ACTION S100_Waiting_for_Start_action:
(* @TEXT_IMPLEMENTATION := 'ST' *)
;
END_ACTION

ACTION S200_AutomaticMode_action:
_FBD_ (* Function Block Diagram *)
_END_FBD_
END_ACTION

ACTION S300_XYZ_PICKnPLACE_SFC_entry:
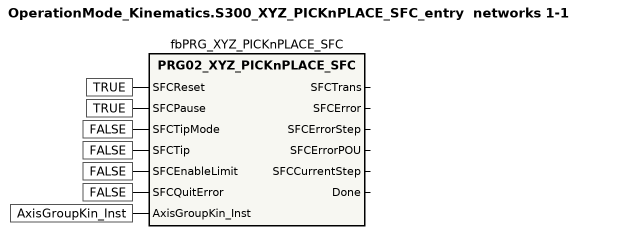
[picture p10: OperationMode_Kinematics.S300_XYZ_PICKnPLACE_SFC_entry (FBD) networks 1-1]
_FBD_ (* Function Block Diagram *)
NETWORK 1
	fbPRG_XYZ_PICKnPLACE_SFC:PRG02_XYZ_PICKnPLACE_SFC(SFCReset: TRUE, SFCPause: TRUE, SFCTipMode: FALSE, SFCTip: FALSE, SFCEnableLimit: FALSE, SFCQuitError: FALSE, AxisGroupKin_Inst: AxisGroupKin_Inst)
_END_FBD_
(* the same logic as Structured Text *)
(* Network 1 *)
fbPRG_XYZ_PICKnPLACE_SFC(SFCReset := TRUE, SFCPause := TRUE, SFCTipMode := FALSE, SFCTip := FALSE, SFCEnableLimit := FALSE, SFCQuitError := FALSE, AxisGroupKin_Inst := AxisGroupKin_Inst);
END_ACTION

ACTION S300_XYZ_PICKnPLACE_SFC_action:
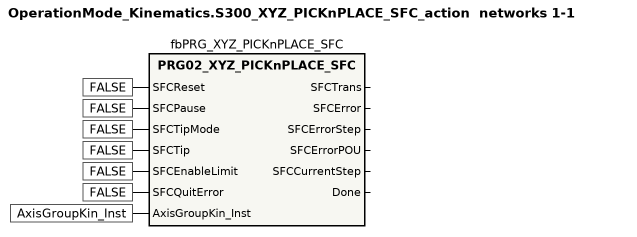
_FBD_ (* Function Block Diagram *)
NETWORK 1
	fbPRG_XYZ_PICKnPLACE_SFC:PRG02_XYZ_PICKnPLACE_SFC(SFCReset: FALSE, SFCPause: FALSE, SFCTipMode: FALSE, SFCTip: FALSE, SFCEnableLimit: FALSE, SFCQuitError: FALSE, AxisGroupKin_Inst: AxisGroupKin_Inst)
_END_FBD_
(* the same logic as Structured Text *)
(* Network 1 *)
fbPRG_XYZ_PICKnPLACE_SFC(SFCReset := FALSE, SFCPause := FALSE, SFCTipMode := FALSE, SFCTip := FALSE, SFCEnableLimit := FALSE, SFCQuitError := FALSE, AxisGroupKin_Inst := AxisGroupKin_Inst);
END_ACTION

ACTION S350_XYZ_TARG_LIN_CIRC_ST_entry:
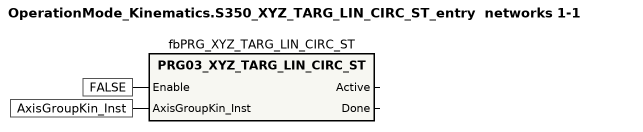
_FBD_ (* Function Block Diagram *)
NETWORK 1
	fbPRG_XYZ_TARG_LIN_CIRC_ST:PRG03_XYZ_TARG_LIN_CIRC_ST(Enable: FALSE, AxisGroupKin_Inst: AxisGroupKin_Inst)
_END_FBD_
(* the same logic as Structured Text *)
(* Network 1 *)
fbPRG_XYZ_TARG_LIN_CIRC_ST(Enable := FALSE, AxisGroupKin_Inst := AxisGroupKin_Inst);
END_ACTION

ACTION S350_XYZ_TARG_LIN_CIRC_ST_action:
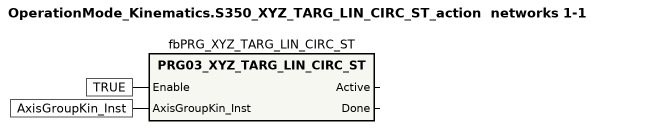
_FBD_ (* Function Block Diagram *)
NETWORK 1
	fbPRG_XYZ_TARG_LIN_CIRC_ST:PRG03_XYZ_TARG_LIN_CIRC_ST(Enable: TRUE, AxisGroupKin_Inst: AxisGroupKin_Inst)
_END_FBD_
(* the same logic as Structured Text *)
(* Network 1 *)
fbPRG_XYZ_TARG_LIN_CIRC_ST(Enable := TRUE, AxisGroupKin_Inst := AxisGroupKin_Inst);
END_ACTION

ACTION S400_XYZ_TARG_LIN_CIRC_SFC_entry:
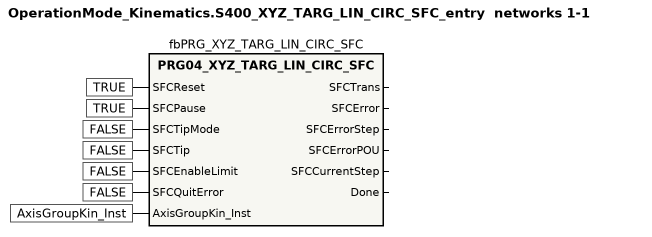
_FBD_ (* Function Block Diagram *)
NETWORK 1
	fbPRG_XYZ_TARG_LIN_CIRC_SFC:PRG04_XYZ_TARG_LIN_CIRC_SFC(SFCReset: TRUE, SFCPause: TRUE, SFCTipMode: FALSE, SFCTip: FALSE, SFCEnableLimit: FALSE, SFCQuitError: FALSE, AxisGroupKin_Inst: AxisGroupKin_Inst)
_END_FBD_
(* the same logic as Structured Text *)
(* Network 1 *)
fbPRG_XYZ_TARG_LIN_CIRC_SFC(SFCReset := TRUE, SFCPause := TRUE, SFCTipMode := FALSE, SFCTip := FALSE, SFCEnableLimit := FALSE, SFCQuitError := FALSE, AxisGroupKin_Inst := AxisGroupKin_Inst);
END_ACTION

ACTION S400_XYZ_TARG_LIN_CIRC_SFC_action:
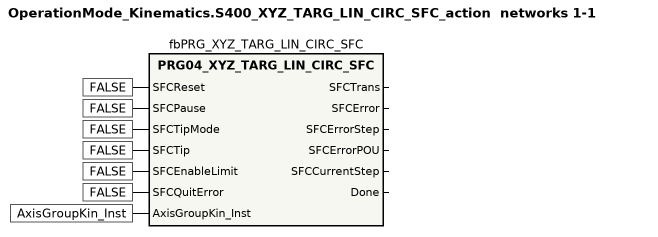
_FBD_ (* Function Block Diagram *)
NETWORK 1
	fbPRG_XYZ_TARG_LIN_CIRC_SFC:PRG04_XYZ_TARG_LIN_CIRC_SFC(SFCReset: FALSE, SFCPause: FALSE, SFCTipMode: FALSE, SFCTip: FALSE, SFCEnableLimit: FALSE, SFCQuitError: FALSE, AxisGroupKin_Inst: AxisGroupKin_Inst)
_END_FBD_
(* the same logic as Structured Text *)
(* Network 1 *)
fbPRG_XYZ_TARG_LIN_CIRC_SFC(SFCReset := FALSE, SFCPause := FALSE, SFCTipMode := FALSE, SFCTip := FALSE, SFCEnableLimit := FALSE, SFCQuitError := FALSE, AxisGroupKin_Inst := AxisGroupKin_Inst);
END_ACTION

ACTION S450_XYZ_USER_ST_entry:
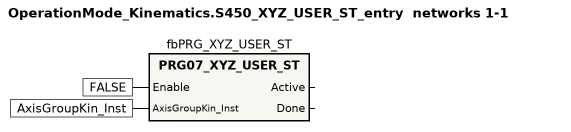
_FBD_ (* Function Block Diagram *)
NETWORK 1
	fbPRG_XYZ_USER_ST:PRG07_XYZ_USER_ST(Enable: FALSE, AxisGroupKin_Inst: AxisGroupKin_Inst)
_END_FBD_
(* the same logic as Structured Text *)
(* Network 1 *)
fbPRG_XYZ_USER_ST(Enable := FALSE, AxisGroupKin_Inst := AxisGroupKin_Inst);
END_ACTION

ACTION S450_XYZ_USER_ST_action:
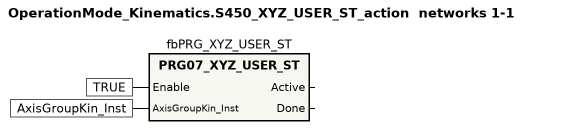
_FBD_ (* Function Block Diagram *)
NETWORK 1
	fbPRG_XYZ_USER_ST:PRG07_XYZ_USER_ST(Enable: TRUE, AxisGroupKin_Inst: AxisGroupKin_Inst)
_END_FBD_
(* the same logic as Structured Text *)
(* Network 1 *)
fbPRG_XYZ_USER_ST(Enable := TRUE, AxisGroupKin_Inst := AxisGroupKin_Inst);
END_ACTION

ACTION S500_XYZ_USER_SFC_entry:
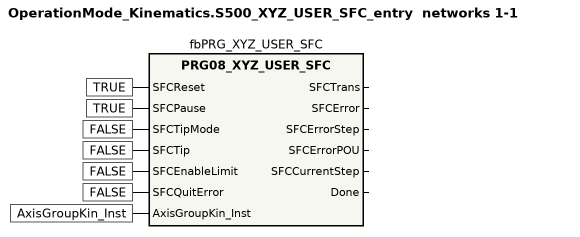
_FBD_ (* Function Block Diagram *)
NETWORK 1
	fbPRG_XYZ_USER_SFC:PRG08_XYZ_USER_SFC(SFCReset: TRUE, SFCPause: TRUE, SFCTipMode: FALSE, SFCTip: FALSE, SFCEnableLimit: FALSE, SFCQuitError: FALSE, AxisGroupKin_Inst: AxisGroupKin_Inst)
_END_FBD_
(* the same logic as Structured Text *)
(* Network 1 *)
fbPRG_XYZ_USER_SFC(SFCReset := TRUE, SFCPause := TRUE, SFCTipMode := FALSE, SFCTip := FALSE, SFCEnableLimit := FALSE, SFCQuitError := FALSE, AxisGroupKin_Inst := AxisGroupKin_Inst);
END_ACTION

ACTION S500_XYZ_USER_SFC_action:
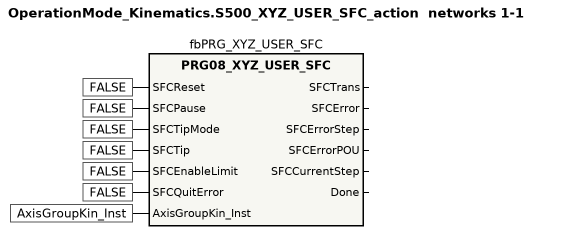
_FBD_ (* Function Block Diagram *)
NETWORK 1
	fbPRG_XYZ_USER_SFC:PRG08_XYZ_USER_SFC(SFCReset: FALSE, SFCPause: FALSE, SFCTipMode: FALSE, SFCTip: FALSE, SFCEnableLimit: FALSE, SFCQuitError: FALSE, AxisGroupKin_Inst: AxisGroupKin_Inst)
_END_FBD_
(* the same logic as Structured Text *)
(* Network 1 *)
fbPRG_XYZ_USER_SFC(SFCReset := FALSE, SFCPause := FALSE, SFCTipMode := FALSE, SFCTip := FALSE, SFCEnableLimit := FALSE, SFCQuitError := FALSE, AxisGroupKin_Inst := AxisGroupKin_Inst);
END_ACTION

ACTION S550_XYZ_FillQueue_LIN3D_with_Array_ST_entry:
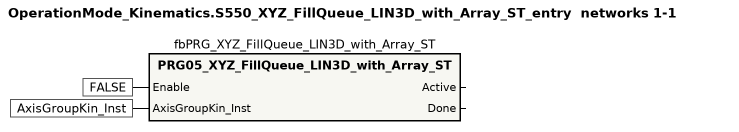
_FBD_ (* Function Block Diagram *)
NETWORK 1
	fbPRG_XYZ_FillQueue_LIN3D_with_Array_ST:PRG05_XYZ_FillQueue_LIN3D_with_Array_ST(Enable: FALSE, AxisGroupKin_Inst: AxisGroupKin_Inst)
_END_FBD_
(* the same logic as Structured Text *)
(* Network 1 *)
fbPRG_XYZ_FillQueue_LIN3D_with_Array_ST(Enable := FALSE, AxisGroupKin_Inst := AxisGroupKin_Inst);
END_ACTION

ACTION S550_XYZ_FillQueue_LIN3D_with_Array_ST_action:
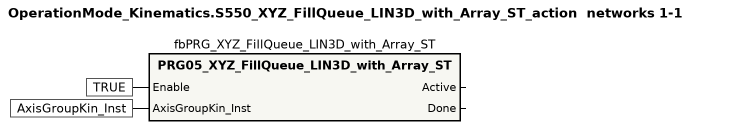
_FBD_ (* Function Block Diagram *)
NETWORK 1
	fbPRG_XYZ_FillQueue_LIN3D_with_Array_ST:PRG05_XYZ_FillQueue_LIN3D_with_Array_ST(Enable: TRUE, AxisGroupKin_Inst: AxisGroupKin_Inst)
_END_FBD_
(* the same logic as Structured Text *)
(* Network 1 *)
fbPRG_XYZ_FillQueue_LIN3D_with_Array_ST(Enable := TRUE, AxisGroupKin_Inst := AxisGroupKin_Inst);
END_ACTION

ACTION S600_XYZ_FillQueue_LIN3D_with_Array_SFC_entry:
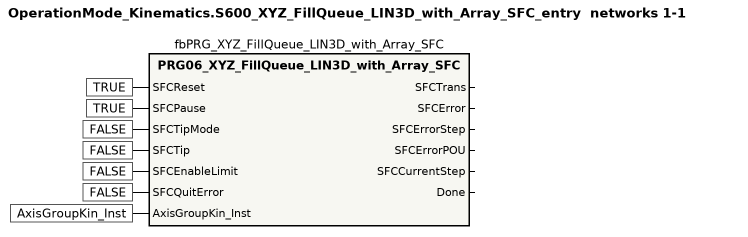
_FBD_ (* Function Block Diagram *)
NETWORK 1
	fbPRG_XYZ_FillQueue_LIN3D_with_Array_SFC:PRG06_XYZ_FillQueue_LIN3D_with_Array_SFC(SFCReset: TRUE, SFCPause: TRUE, SFCTipMode: FALSE, SFCTip: FALSE, SFCEnableLimit: FALSE, SFCQuitError: FALSE, AxisGroupKin_Inst: AxisGroupKin_Inst)
_END_FBD_
(* the same logic as Structured Text *)
(* Network 1 *)
fbPRG_XYZ_FillQueue_LIN3D_with_Array_SFC(SFCReset := TRUE, SFCPause := TRUE, SFCTipMode := FALSE, SFCTip := FALSE, SFCEnableLimit := FALSE, SFCQuitError := FALSE, AxisGroupKin_Inst := AxisGroupKin_Inst);
END_ACTION

ACTION S600_XYZ_FillQueue_LIN3D_with_Array_SFC_action:
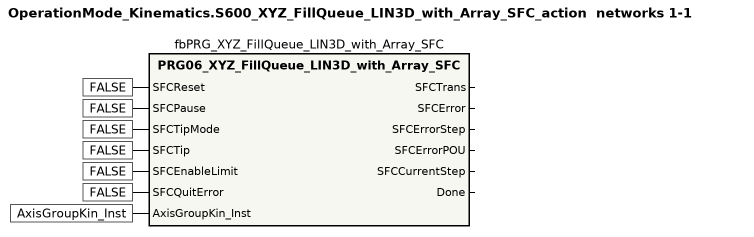
_FBD_ (* Function Block Diagram *)
NETWORK 1
	fbPRG_XYZ_FillQueue_LIN3D_with_Array_SFC:PRG06_XYZ_FillQueue_LIN3D_with_Array_SFC(SFCReset: FALSE, SFCPause: FALSE, SFCTipMode: FALSE, SFCTip: FALSE, SFCEnableLimit: FALSE, SFCQuitError: FALSE, AxisGroupKin_Inst: AxisGroupKin_Inst)
_END_FBD_
(* the same logic as Structured Text *)
(* Network 1 *)
fbPRG_XYZ_FillQueue_LIN3D_with_Array_SFC(SFCReset := FALSE, SFCPause := FALSE, SFCTipMode := FALSE, SFCTip := FALSE, SFCEnableLimit := FALSE, SFCQuitError := FALSE, AxisGroupKin_Inst := AxisGroupKin_Inst);
END_ACTION

ACTION S250_XYZ_PICKnPLACE_ST_entry:
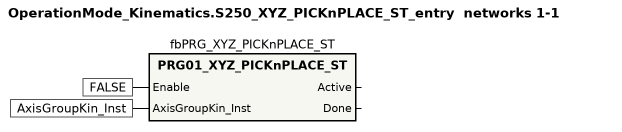
_FBD_ (* Function Block Diagram *)
NETWORK 1
	fbPRG_XYZ_PICKnPLACE_ST:PRG01_XYZ_PICKnPLACE_ST(Enable: FALSE, AxisGroupKin_Inst: AxisGroupKin_Inst)
_END_FBD_
(* the same logic as Structured Text *)
(* Network 1 *)
fbPRG_XYZ_PICKnPLACE_ST(Enable := FALSE, AxisGroupKin_Inst := AxisGroupKin_Inst);
END_ACTION

ACTION S250_XYZ_PICKnPLACE_ST_action:
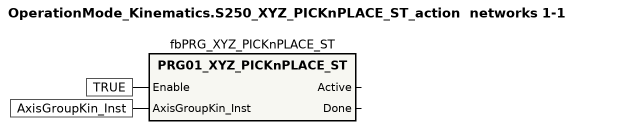
_FBD_ (* Function Block Diagram *)
NETWORK 1
	fbPRG_XYZ_PICKnPLACE_ST:PRG01_XYZ_PICKnPLACE_ST(Enable: TRUE, AxisGroupKin_Inst: AxisGroupKin_Inst)
_END_FBD_
(* the same logic as Structured Text *)
(* Network 1 *)
fbPRG_XYZ_PICKnPLACE_ST(Enable := TRUE, AxisGroupKin_Inst := AxisGroupKin_Inst);
END_ACTION

TRANSITION NOT referenced:
_FBD_ (* Function Block Diagram *)
NETWORK 1
	AND(AxisGroupKin_Inst.Out.General.Inverter.Connected[0], NOT AxisGroupKin_Inst.Out.General.Inverter.Referenced[0])
_END_FBD_
END_TRANSITION

TRANSITION referenced:
_FBD_ (* Function Block Diagram *)
NETWORK 1
	AND(AxisGroupKin_Inst.Out.General.Inverter.Connected[0], AxisGroupKin_Inst.Out.General.Inverter.Referenced[0])
_END_FBD_
END_TRANSITION

TRANSITION Homing done:
_FBD_ (* Function Block Diagram *)
NETWORK 1
	AND(AxisGroupKin_Inst.Out.General.Inverter.Connected[0], AxisGroupKin_Inst.Out.General.Inverter.Referenced[0])
_END_FBD_
END_TRANSITION

TRANSITION Automatic Mode:
_FBD_ (* Function Block Diagram *)
NETWORK 1
	AxisGroupKin_Inst.Out.General.Kin.Ready
_END_FBD_
(* the same logic as Structured Text *)
(* Network 1 *)
Automatic_Mode := AxisGroupKin_Inst.Out.General.Kin.Ready;
END_TRANSITION

TRANSITION Jog Mode:
_FBD_ (* Function Block Diagram *)
NETWORK 1
	NOT FALSE
_END_FBD_
(* the same logic as Structured Text *)
(* Network 1 *)
Jog_Mode := NOT FALSE;
END_TRANSITION

TRANSITION no Jog Mode:
_FBD_ (* Function Block Diagram *)
NETWORK 1
	FALSE
_END_FBD_
(* the same logic as Structured Text *)
(* Network 1 *)
no_Jog_Mode := FALSE;
END_TRANSITION

TRANSITION Start AND Enabled:
_FBD_ (* Function Block Diagram *)
NETWORK 1
	AND(TRUE, AxisGroupKin_Inst.Out.General.Kin.Ready)
_END_FBD_
END_TRANSITION

TRANSITION PRG1_Pick_and_Place_ST:
_FBD_ (* Function Block Diagram *)
NETWORK 1
	EQ(gKinExamples_Control[InstanceNumber].ProgramNumber, 1)
_END_FBD_
END_TRANSITION

TRANSITION Pick_and_Place_SFC:
_FBD_ (* Function Block Diagram *)
NETWORK 1
	EQ(gKinExamples_Control[InstanceNumber].ProgramNumber, 2)
_END_FBD_
END_TRANSITION

TRANSITION new Mode or Done:
_FBD_ (* Function Block Diagram *)
NETWORK 1
	OR(NE(gKinExamples_Control[InstanceNumber].ProgramNumber, 2), fbPRG_XYZ_PICKnPLACE_SFC.Done)
_END_FBD_
END_TRANSITION

TRANSITION XYZ_TARG_LIN_CIRC_ST:
_FBD_ (* Function Block Diagram *)
NETWORK 1
	EQ(gKinExamples_Control[InstanceNumber].ProgramNumber, 3)
_END_FBD_
END_TRANSITION

TRANSITION new Mode or Done:
_FBD_ (* Function Block Diagram *)
NETWORK 1
	OR(NE(gKinExamples_Control[InstanceNumber].ProgramNumber, 3), fbPRG_XYZ_TARG_LIN_CIRC_ST.Done)
_END_FBD_
END_TRANSITION

TRANSITION XYZ_TARG_LIN_CIRC_SFC:
_FBD_ (* Function Block Diagram *)
NETWORK 1
	EQ(gKinExamples_Control[InstanceNumber].ProgramNumber, 4)
_END_FBD_
END_TRANSITION

TRANSITION new Mode or Done:
_FBD_ (* Function Block Diagram *)
NETWORK 1
	OR(NE(gKinExamples_Control[InstanceNumber].ProgramNumber, 4), fbPRG_XYZ_TARG_LIN_CIRC_SFC.Done)
_END_FBD_
END_TRANSITION

TRANSITION XYZ_USER_ST:
_FBD_ (* Function Block Diagram *)
NETWORK 1
	EQ(gKinExamples_Control[InstanceNumber].ProgramNumber, 7)
_END_FBD_
END_TRANSITION

TRANSITION new Mode or Done:
_FBD_ (* Function Block Diagram *)
NETWORK 1
	OR(NE(gKinExamples_Control[InstanceNumber].ProgramNumber, 7), fbPRG_XYZ_USER_ST.Done)
_END_FBD_
END_TRANSITION

TRANSITION XYZ_USER_SFC:
_FBD_ (* Function Block Diagram *)
NETWORK 1
	EQ(gKinExamples_Control[InstanceNumber].ProgramNumber, 8)
_END_FBD_
END_TRANSITION

TRANSITION new Mode or Done:
_FBD_ (* Function Block Diagram *)
NETWORK 1
	OR(NE(gKinExamples_Control[InstanceNumber].ProgramNumber, 8), fbPRG_XYZ_USER_SFC.Done)
_END_FBD_
END_TRANSITION

TRANSITION FillQueue_LIN3D_with_Array_ST:
_FBD_ (* Function Block Diagram *)
NETWORK 1
	EQ(gKinExamples_Control[InstanceNumber].ProgramNumber, 5)
_END_FBD_
END_TRANSITION

TRANSITION new Mode or Done:
_FBD_ (* Function Block Diagram *)
NETWORK 1
	OR(NE(gKinExamples_Control[InstanceNumber].ProgramNumber, 5), fbPRG_XYZ_FillQueue_LIN3D_with_Array_ST.Done)
_END_FBD_
END_TRANSITION

TRANSITION FillQueue_LIN3D_with_Array_SFC:
_FBD_ (* Function Block Diagram *)
NETWORK 1
	EQ(gKinExamples_Control[InstanceNumber].ProgramNumber, 6)
_END_FBD_
END_TRANSITION

TRANSITION new Mode OR Done:
_FBD_ (* Function Block Diagram *)
NETWORK 1
	OR(NE(gKinExamples_Control[InstanceNumber].ProgramNumber, 6), fbPRG_XYZ_FillQueue_LIN3D_with_Array_SFC.Done)
_END_FBD_
END_TRANSITION

TRANSITION Jog Mode:
_FBD_ (* Function Block Diagram *)
NETWORK 1
	NOT FALSE
_END_FBD_
(* the same logic as Structured Text *)
(* Network 1 *)
Jog_Mode := NOT FALSE;
END_TRANSITION

TRANSITION new Mode or Done:
_FBD_ (* Function Block Diagram *)
NETWORK 1
	OR(NE(gKinExamples_Control[InstanceNumber].ProgramNumber, 1), fbPRG_XYZ_PICKnPLACE_ST.Done)
_END_FBD_
END_TRANSITION
END_FUNCTION_BLOCK

(* POU AxisGroupControl_Kinematics/Examples/PRG01_XYZ_PICKnPLACE_ST, ST *)
(*##############################################################################################################

	IMPORTANT NOTICE:
 	This example is a special and free service that demonstrates only the basic 
	approach to generating a PLC program as a non-binding sample. 
	SEW is not liable for the contents of the sample program.

	Name:			PRG_XYZ_PICKnPLACE_ST
	Job:			Example program		
					Sequence: XYZ_PICKnPLACE_P2 -> P3 -> P4 -> P3 -> P2 -> P1
					
################################################################################################################*)
FUNCTION_BLOCK  PRG01_XYZ_PICKnPLACE_ST
VAR_INPUT
	Enable : BOOL;
END_VAR
VAR_OUTPUT
	Active : BOOL;
	Done : BOOL;
END_VAR
VAR
	nState : INT := 0;
	fbRtrig : R_TRIG;
	i : INT;
END_VAR
VAR_IN_OUT
	AxisGroupKin_Inst											: ST_AxisGroupKin_Instance;
END_VAR
(* Initialisation at rising edge of VAR_INPUT Enable *)
fbRtrig(CLK:=Enable);
IF fbRtrig.Q THEN
	nState := 0;
	Active := TRUE;
END_IF

(* No execution, if Enable = False *)
IF (Enable = FALSE) THEN
	Done := FALSE;
	RETURN;
END_IF


CASE nState OF
0:	(*Start*)
	IF AxisGroupKin.ConfigDataAvailable THEN
		nState := 5;
	END_IF

5:	(* Up *)
	(* Initialize Kinematic Flags*)
	AxisGroupKin_Inst.In.Cp.Settings.PlusTargetCartABC:=FALSE;
	AxisGroupKin_Inst.In.Cp.Settings.UseMasterPosition:=FALSE;

(* TARGET_CART settings *)
	(* Motion Parameters *)
	AxisGroupKin_Inst.In.Target.Cart.Velocity := CART_VEL100;
	AxisGroupKin_Inst.In.Target.Cart.Acceleration := CART_ACC100;
	AxisGroupKin_Inst.In.Target.Cart.Deceleration := CART_DEC100;
	AxisGroupKin_Inst.In.Target.Cart.Jerk:=CART_Jerk100;
	AxisGroupKin_Inst.In.Target.Synchronization:= KIN_NO_SYNC;
	(* Coordinate System *)
	AxisGroupKin_Inst.In.Target.CoordSys:=KIN_KCS;

	AxisGroupKin_Inst.In.General.Mode := KIN_TARGET_CART;

	AxisGroupKin_Inst.In.Target.Position := XYZ_PICKnPLACE_P2;

	IF (MC_KinInProximity(Threshold := XYZ_PICKnPLACE_BlendingDistance,
			Position := AxisGroupKin_Inst.In.Target.Position,
			CoordSys := AxisGroupKin_Inst.In.Target.CoordSys,
			Dimension := 2#0000_0111, ActPos := AxisGroupKin_Inst.Out.General.Position)) THEN
		nState := 10;
	END_IF
	AxisGroupKin_Inst.In.Simu3D.Ctrl.Pen_TCP_WCS:=TRUE;

10:	(* Side *)
	AxisGroupKin_Inst.In.Target.Position := XYZ_PICKnPLACE_P3;
	IF (MC_KinInProximity(Threshold := XYZ_PICKnPLACE_BlendingDistance,
			Position := AxisGroupKin_Inst.In.Target.Position,
			CoordSys := AxisGroupKin_Inst.In.Target.CoordSys,
			Dimension := 2#0000_0111, ActPos := AxisGroupKin_Inst.Out.General.Position)) THEN
		nState := 20;
	END_IF

20:	(* Down *)
	AxisGroupKin_Inst.In.Target.Position := XYZ_PICKnPLACE_P4;
	IF (MC_KinInProximity(Threshold := 0.0,
			Position := AxisGroupKin_Inst.In.Target.Position,
			CoordSys := AxisGroupKin_Inst.In.Target.CoordSys,
			Dimension := 2#0000_0111, ActPos := AxisGroupKin_Inst.Out.General.Position)
			AND AxisGroupKin_Inst.Out.General.Standstill.ActCoordSys) THEN
		nState :=30;
	END_IF

30:	(* Up *)
	AxisGroupKin_Inst.In.Target.Position := XYZ_PICKnPLACE_P3;
	IF (MC_KinInProximity(Threshold := XYZ_PICKnPLACE_BlendingDistance,
			Position := AxisGroupKin_Inst.In.Target.Position,
			CoordSys := AxisGroupKin_Inst.In.Target.CoordSys,
			Dimension := 2#0000_0111, ActPos := AxisGroupKin_Inst.Out.General.Position)) THEN
		nState := 40;
	END_IF

40:	(* Side *)
	AxisGroupKin_Inst.In.Target.Position := XYZ_PICKnPLACE_P2;
	IF (MC_KinInProximity(Threshold := XYZ_PICKnPLACE_BlendingDistance,
			Position := AxisGroupKin_Inst.In.Target.Position,
			CoordSys := AxisGroupKin_Inst.In.Target.CoordSys,
			Dimension := 2#0000_0111, ActPos := AxisGroupKin_Inst.Out.General.Position)) THEN
		nState := 50;
	END_IF

50:	(* Down *)
	AxisGroupKin_Inst.In.Target.Position := XYZ_PICKnPLACE_P1;
	IF (MC_KinInProximity(Threshold := 0.0,
			Position := AxisGroupKin_Inst.In.Target.Position,
			CoordSys := AxisGroupKin_Inst.In.Target.CoordSys,
			Dimension := 2#0000_0111, ActPos := AxisGroupKin_Inst.Out.General.Position)
			AND AxisGroupKin_Inst.Out.General.Standstill.ActCoordSys) THEN
		AxisGroupKin_Inst.In.Simu3D.Ctrl.Pen_TCP_WCS:=FALSE;
		Done := TRUE;
		Active := FALSE;
	END_IF

ELSE
;

END_CASE
END_FUNCTION_BLOCK

(* POU AxisGroupControl_Kinematics/Examples/PRG02_XYZ_PICKnPLACE_SFC, SFC *)
(*##############################################################################################################

	IMPORTANT NOTICE:
 	This example is a special and free service that demonstrates only the basic 
	approach to generating a PLC program as a non-binding sample. 
	SEW is not liable for the contents of the sample program.

	Name:			PRG_XYZ_PICKnPLACE_SFC
	Job:			Example program		
					Sequence: XYZ_PICKnPLACE_P2 -> P3 -> P4 -> P3 -> P2 -> P1	

################################################################################################################*)
FUNCTION_BLOCK PRG02_XYZ_PICKnPLACE_SFC
VAR_INPUT
	SFCReset:BOOL;
	(*SFCInit:BOOL;*)
	SFCPause:BOOL;

	SFCTipMode:BOOL;
	SFCTip:BOOL;
	SFCEnableLimit:BOOL;
	SFCQuitError:BOOL;
END_VAR
VAR_OUTPUT
	SFCTrans:BOOL;
	SFCError:BOOL;
	SFCErrorStep:STRING;
	SFCErrorPOU:STRING;
	SFCCurrentStep:STRING;
	Done:BOOL;
END_VAR
VAR

END_VAR
VAR_IN_OUT
	AxisGroupKin_Inst											: ST_AxisGroupKin_Instance;
END_VAR
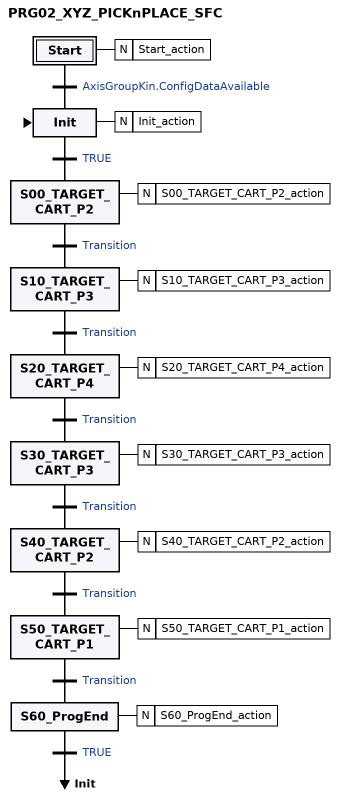
INITIAL_STEP Start:
	Start_action(N);
END_STEP
TRANSITION FROM Start TO Init := AxisGroupKin.ConfigDataAvailable;
END_TRANSITION
STEP Init:
	Init_action(N);
END_STEP
TRANSITION FROM Init TO S00_TARGET_CART_P2 := TRUE;
END_TRANSITION
STEP S00_TARGET_CART_P2:
	S00_TARGET_CART_P2_action(N);
END_STEP
TRANSITION FROM S00_TARGET_CART_P2 TO S10_TARGET_CART_P3 := Transition;
END_TRANSITION
STEP S10_TARGET_CART_P3:
	S10_TARGET_CART_P3_action(N);
END_STEP
TRANSITION FROM S10_TARGET_CART_P3 TO S20_TARGET_CART_P4 := Transition;
END_TRANSITION
STEP S20_TARGET_CART_P4:
	S20_TARGET_CART_P4_action(N);
END_STEP
TRANSITION FROM S20_TARGET_CART_P4 TO S30_TARGET_CART_P3 := Transition;
END_TRANSITION
STEP S30_TARGET_CART_P3:
	S30_TARGET_CART_P3_action(N);
END_STEP
TRANSITION FROM S30_TARGET_CART_P3 TO S40_TARGET_CART_P2 := Transition;
END_TRANSITION
STEP S40_TARGET_CART_P2:
	S40_TARGET_CART_P2_action(N);
END_STEP
TRANSITION FROM S40_TARGET_CART_P2 TO S50_TARGET_CART_P1 := Transition;
END_TRANSITION
STEP S50_TARGET_CART_P1:
	S50_TARGET_CART_P1_action(N);
END_STEP
TRANSITION FROM S50_TARGET_CART_P1 TO S60_ProgEnd := Transition;
END_TRANSITION
STEP S60_ProgEnd:
	S60_ProgEnd_action(N);
END_STEP
TRANSITION FROM S60_ProgEnd TO Init := TRUE;
END_TRANSITION

ACTION Start_action:
Done:=FALSE;
END_ACTION

ACTION Init_action:
(* Initialize Kinematic Flags*)
	AxisGroupKin_Inst.In.Cp.Settings.PlusTargetCartABC:=FALSE;
	AxisGroupKin_Inst.In.Cp.Settings.UseMasterPosition:=FALSE;

(* TARGET_CART settings *)
	(* Motion Parameters *)
	AxisGroupKin_Inst.In.Target.Cart.Velocity := CART_VEL100;
	AxisGroupKin_Inst.In.Target.Cart.Acceleration := CART_ACC100;
	AxisGroupKin_Inst.In.Target.Cart.Deceleration := CART_DEC100;
	AxisGroupKin_Inst.In.Target.Cart.Jerk := CART_Jerk100;
	AxisGroupKin_Inst.In.Target.Synchronization := KIN_NO_SYNC;
	(* Coordinate System *)
	AxisGroupKin_Inst.In.Target.CoordSys := KIN_KCS;

	AxisGroupKin_Inst.In.General.Mode := KIN_TARGET_CART;
END_ACTION

ACTION S00_TARGET_CART_P2_action:
AxisGroupKin_Inst.In.Target.Position := XYZ_PICKnPLACE_P2;
END_ACTION

ACTION S10_TARGET_CART_P3_action:
AxisGroupKin_Inst.In.Target.Position := XYZ_PICKnPLACE_P3;
END_ACTION

ACTION S20_TARGET_CART_P4_action:
AxisGroupKin_Inst.In.Target.Position := XYZ_PICKnPLACE_P4;
END_ACTION

ACTION S30_TARGET_CART_P3_action:
AxisGroupKin_Inst.In.Target.Position := XYZ_PICKnPLACE_P3;
END_ACTION

ACTION S40_TARGET_CART_P2_action:
AxisGroupKin_Inst.In.Target.Position := XYZ_PICKnPLACE_P2;
END_ACTION

ACTION S50_TARGET_CART_P1_action:
AxisGroupKin_Inst.In.Target.Position := XYZ_PICKnPLACE_P1;
END_ACTION

ACTION S60_ProgEnd_action:
Done:=TRUE;
END_ACTION

TRANSITION Transition:
MC_KinInProximity(Threshold := XYZ_PICKnPLACE_BlendingDistance,
			Position := AxisGroupKin_Inst.In.Target.Position,
			CoordSys := AxisGroupKin_Inst.In.Target.CoordSys,
			Dimension := 2#0000_0111, ActPos := AxisGroupKin_Inst.Out.General.Position)
END_TRANSITION

TRANSITION Transition:
MC_KinInProximity(Threshold := XYZ_PICKnPLACE_BlendingDistance,
			Position := AxisGroupKin_Inst.In.Target.Position,
			CoordSys := AxisGroupKin_Inst.In.Target.CoordSys,
			Dimension := 2#0000_0111, ActPos := AxisGroupKin_Inst.Out.General.Position)
END_TRANSITION

TRANSITION Transition:
MC_KinInProximity(Threshold := 0.0,
			Position := AxisGroupKin_Inst.In.Target.Position,
			CoordSys := AxisGroupKin_Inst.In.Target.CoordSys,
			Dimension := 2#0000_0111, ActPos := AxisGroupKin_Inst.Out.General.Position)
AND
AxisGroupKin_Inst.Out.General.Standstill.ActCoordSys
END_TRANSITION

TRANSITION Transition:
MC_KinInProximity(Threshold := XYZ_PICKnPLACE_BlendingDistance,
			Position := AxisGroupKin_Inst.In.Target.Position,
			CoordSys := AxisGroupKin_Inst.In.Target.CoordSys,
			Dimension := 2#0000_0111, ActPos := AxisGroupKin_Inst.Out.General.Position)
END_TRANSITION

TRANSITION Transition:
MC_KinInProximity(Threshold := XYZ_PICKnPLACE_BlendingDistance,
			Position := AxisGroupKin_Inst.In.Target.Position,
			CoordSys := AxisGroupKin_Inst.In.Target.CoordSys,
			Dimension := 2#0000_0111, ActPos := AxisGroupKin_Inst.Out.General.Position)
END_TRANSITION

TRANSITION Transition:
MC_KinInProximity(Threshold := 0.0,
			Position := AxisGroupKin_Inst.In.Target.Position,
			CoordSys := AxisGroupKin_Inst.In.Target.CoordSys,
			Dimension := 2#0000_0111, ActPos := AxisGroupKin_Inst.Out.General.Position)
AND
AxisGroupKin_Inst.Out.General.Standstill.ActCoordSys
END_TRANSITION
END_FUNCTION_BLOCK

(* POU AxisGroupControl_Kinematics/Examples/PRG03_XYZ_TARG_LIN_CIRC_ST, ST *)
(*##############################################################################################################

	IMPORTANT NOTICE:
 	This example is a special and free service that demonstrates only the basic 
	approach to generating a PLC program as a non-binding sample. 
	SEW is not liable for the contents of the sample program.

	Name:			PRG_XYZ_TARG_LIN_CIRC_ST
	Job:			Example program			
					Sequence: TARGET_CART to XYZ_TARG_LIN_CIRC_P1 -> LIN_XY to P2 -> CIRC_XZ with R3/A3 -> LIN_3D to P4 -> LIN_XY to P1

################################################################################################################*)
FUNCTION_BLOCK PRG03_XYZ_TARG_LIN_CIRC_ST
VAR_INPUT
	Enable : BOOL;
END_VAR
VAR_OUTPUT
	Active : BOOL;
	Done : BOOL;
END_VAR
VAR
	nState : INT;
	fbRtrig : R_TRIG;
END_VAR
VAR_IN_OUT
	AxisGroupKin_Inst											: ST_AxisGroupKin_Instance;
END_VAR
(* Initialisation at rising edge of VAR_INPUT Enable *)
fbRtrig(CLK:=Enable);
IF fbRtrig.Q THEN
	nState	:= 0;
	Active := TRUE;
END_IF

(* No execution, if Enable = False *)
IF NOT Enable THEN
	Done := FALSE;
	RETURN;
END_IF


CASE nState OF
0:	(*Start*)
	IF AxisGroupKin.ConfigDataAvailable THEN
		nState := 5;
	END_IF
5:	(* TARGET_CART to XYZ_TARG_LIN_CIRC_P1 *)
	(* Initialize Kinematic Flags*)
	AxisGroupKin_Inst.In.Cp.Settings.PlusTargetCartABC:=FALSE;
	AxisGroupKin_Inst.In.Cp.Settings.UseMasterPosition:=FALSE;

(* TARGET_CART settings *)
	(* Motion Parameters *)
	AxisGroupKin_Inst.In.Target.Cart.Acceleration := CART_ACC50;
	AxisGroupKin_Inst.In.Target.Cart.Deceleration := CART_DEC50;
	AxisGroupKin_Inst.In.Target.Cart.Velocity := CART_VEL50;
	AxisGroupKin_Inst.In.Target.Cart.Jerk:=CART_Jerk100;
	AxisGroupKin_Inst.In.Target.Synchronization:= KIN_NO_SYNC;
	(* Coordinate System *)
	AxisGroupKin_Inst.In.Target.CoordSys:=KIN_KCS;

	AxisGroupKin_Inst.In.General.Mode := KIN_TARGET_CART;

	AxisGroupKin_Inst.In.Target.Position := XYZ_TARG_LIN_CIRC_P1;
	IF (MC_KinInProximity(Threshold := 0.0,
			Position := AxisGroupKin_Inst.In.Target.Position,
			CoordSys := AxisGroupKin_Inst.In.Target.CoordSys,
			Dimension := 2#0000_0111, ActPos := AxisGroupKin_Inst.Out.General.Position)
			AND AxisGroupKin_Inst.Out.General.Standstill.ActCoordSys) THEN
		nState := 10;
	END_IF

10:	(* Straight line to XYZ_TARG_LIN_CIRC_P2, as soon as XYZ_TARG_LIN_CIRC_P1 has been reached *)

		AxisGroupKin_Inst.In.General.Mode := KIN_LIN_XY;
		AxisGroupKin_Inst.In.Cp.Segment.Position := XYZ_TARG_LIN_CIRC_P2;
(* CP motion parameters *)
		(* settings for whole path / all segments *)
		AxisGroupKin_Inst.In.Cp.Path.VelocityPercentage:=100;
		AxisGroupKin_Inst.In.Cp.Path.FidelityPercentage :=100;
		(* Settings for the segment, which should be added to the queue *)
		AxisGroupKin_Inst.In.Cp.Segment.Translation.Velocity := 1000;
		AxisGroupKin_Inst.In.Cp.Segment.Translation.Acceleration := 100;
		AxisGroupKin_Inst.In.Cp.Segment.Translation.Deceleration := 100;
		AxisGroupKin_Inst.In.Cp.Segment.Translation.Jerk := 100;
		AxisGroupKin_Inst.In.Cp.Segment.Blending.Distance := 50;
		AxisGroupKin_Inst.In.Cp.Segment.Blending.LimitationPercentage := 50;

		AxisGroupKin_Inst.In.Cp.Segment.ID := AxisGroupKin_Inst.In.Cp.Segment.ID + 1;	(* Change the SegmentID to add the segment to the queue *)

		AxisGroupKin_Inst.In.Simu3D.Ctrl.Pen_TCP_WCS := TRUE;

		nState := 20;

20:	(* A circle section is written into the queue directly after the straight line *)
	IF (AxisGroupKin_Inst.Out.Cp.Queue.LastMappedSegID = AxisGroupKin_Inst.In.Cp.Segment.ID) THEN (* Wait until the segment was added to the queue; this is not required if FB_KinControl is executed in the same task *)
		AxisGroupKin_Inst.In.General.Mode := KIN_CIRC_ZX;
		(* Parameters to define the circle *)
		AxisGroupKin_Inst.In.Cp.Segment.Circ.Mode := KIN_RADIUS_ANGLE;	(* Define the circle with the radius and angle *)
		AxisGroupKin_Inst.In.Cp.Segment.Circ.Direction := KIN_CW;	(* Draw circle ClockWise *)
		AxisGroupKin_Inst.In.Cp.Segment.Circ.Radius := XYZ_TARG_LIN_CIRC_R3;
		AxisGroupKin_Inst.In.Cp.Segment.Circ.Angle := XYZ_TARG_LIN_CIRC_A3;


		AxisGroupKin_Inst.In.Cp.Segment.ID := AxisGroupKin_Inst.In.Cp.Segment.ID + 1;
		nState := 30;
	END_IF

30:	(* A Straight line to XYZ_TARG_LIN_CIRC_P4 is written into the queue directly after the circle section
		-> Blending to the straight line is performed automatically *)
	IF (AxisGroupKin_Inst.Out.Cp.Queue.LastMappedSegID = AxisGroupKin_Inst.In.Cp.Segment.ID) THEN
		AxisGroupKin_Inst.In.General.Mode := KIN_LIN_3D;
		AxisGroupKin_Inst.In.Cp.Segment.Position := XYZ_TARG_LIN_CIRC_P4;


		AxisGroupKin_Inst.In.Cp.Segment.ID := AxisGroupKin_Inst.In.Cp.Segment.ID + 1;
		nState := 40;
	END_IF

40:	(* Straight line to XYZ_TARG_LIN_CIRC_P1 is written into the queue directly after the previous straight line
		-> Blending to the straight line is performed automatically *)
	IF (AxisGroupKin_Inst.Out.Cp.Queue.LastMappedSegID = AxisGroupKin_Inst.In.Cp.Segment.ID) THEN
		AxisGroupKin_Inst.In.General.Mode := KIN_LIN_XY;
		AxisGroupKin_Inst.In.Cp.Segment.Position := XYZ_TARG_LIN_CIRC_P1;


		AxisGroupKin_Inst.In.Cp.Segment.ID := AxisGroupKin_Inst.In.Cp.Segment.ID + 1;
		nState := 50;
	END_IF

50:	(* Program end, as soon as XYZ_TARG_LIN_CIRC_P1 has been reached *)
	IF (AxisGroupKin_Inst.Out.Cp.Path.EndReached)
	AND (AxisGroupKin_Inst.Out.Cp.Queue.LastMappedSegID = AxisGroupKin_Inst.In.Cp.Segment.ID) THEN
		Done := TRUE;
		Active := FALSE;
		AxisGroupKin_Inst.In.Simu3D.Ctrl.Pen_TCP_WCS := FALSE;
	END_IF

ELSE
;

END_CASE
END_FUNCTION_BLOCK

(* POU AxisGroupControl_Kinematics/Examples/PRG04_XYZ_TARG_LIN_CIRC_SFC, SFC *)
(*##############################################################################################################

	IMPORTANT NOTICE:
 	This example is a special and free service that demonstrates only the basic 
	approach to generating a PLC program as a non-binding sample. 
	SEW is not liable for the contents of the sample program.

	Name:			PRG_XYZ_TARG_LIN_CIRC_SFC
	Job:			Example program			
					Sequence: TARGET_CART to XYZ_TARG_LIN_CIRC_P1 -> LIN_XY to P2 -> CIRC_XZ with R3/A3 -> LIN_3D to P4 -> LIN_XY to P1

################################################################################################################*)
FUNCTION_BLOCK PRG04_XYZ_TARG_LIN_CIRC_SFC
VAR_INPUT
	SFCReset:BOOL;
	(*SFCInit:BOOL;*)
	SFCPause:BOOL;

	SFCTipMode:BOOL;
	SFCTip:BOOL;
	SFCEnableLimit:BOOL;
	SFCQuitError:BOOL;

END_VAR
VAR_OUTPUT
	SFCTrans:BOOL;
	SFCError:BOOL;
	SFCErrorStep:STRING;
	SFCErrorPOU:STRING;
(*	SFCErrorAnalyzation:STRING;*)
	SFCCurrentStep:STRING;
	Done:BOOL;
END_VAR
VAR

END_VAR
VAR_IN_OUT
	AxisGroupKin_Inst											: ST_AxisGroupKin_Instance;
END_VAR
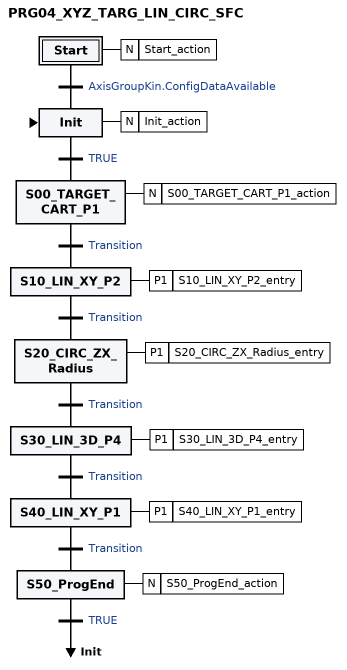
INITIAL_STEP Start:
	Start_action(N);
END_STEP
TRANSITION FROM Start TO Init := AxisGroupKin.ConfigDataAvailable;
END_TRANSITION
STEP Init:
	Init_action(N);
END_STEP
TRANSITION FROM Init TO S00_TARGET_CART_P1 := TRUE;
END_TRANSITION
STEP S00_TARGET_CART_P1:
	S00_TARGET_CART_P1_action(N);
END_STEP
TRANSITION FROM S00_TARGET_CART_P1 TO S10_LIN_XY_P2 := Transition;
END_TRANSITION
STEP S10_LIN_XY_P2:
	S10_LIN_XY_P2_entry(P1);
END_STEP
TRANSITION FROM S10_LIN_XY_P2 TO S20_CIRC_ZX_Radius := Transition;
END_TRANSITION
STEP S20_CIRC_ZX_Radius:
	S20_CIRC_ZX_Radius_entry(P1);
END_STEP
TRANSITION FROM S20_CIRC_ZX_Radius TO S30_LIN_3D_P4 := Transition;
END_TRANSITION
STEP S30_LIN_3D_P4:
	S30_LIN_3D_P4_entry(P1);
END_STEP
TRANSITION FROM S30_LIN_3D_P4 TO S40_LIN_XY_P1 := Transition;
END_TRANSITION
STEP S40_LIN_XY_P1:
	S40_LIN_XY_P1_entry(P1);
END_STEP
TRANSITION FROM S40_LIN_XY_P1 TO S50_ProgEnd := Transition;
END_TRANSITION
STEP S50_ProgEnd:
	S50_ProgEnd_action(N);
END_STEP
TRANSITION FROM S50_ProgEnd TO Init := TRUE;
END_TRANSITION

ACTION Start_action:
Done:=FALSE;
END_ACTION

ACTION Init_action:
(* Initialize Kinematic Flags*)
	AxisGroupKin_Inst.In.Cp.Settings.PlusTargetCartABC:=FALSE;
	AxisGroupKin_Inst.In.Cp.Settings.UseMasterPosition:=FALSE;

(* TARGET_CART settings *)
	(* Motion Parameters *)
	AxisGroupKin_Inst.In.Target.Cart.Acceleration := CART_ACC50;
	AxisGroupKin_Inst.In.Target.Cart.Deceleration := CART_DEC50;
	AxisGroupKin_Inst.In.Target.Cart.Velocity := CART_VEL50;
	AxisGroupKin_Inst.In.Target.Cart.Jerk:=CART_Jerk100;
	AxisGroupKin_Inst.In.Target.Synchronization:= KIN_NO_SYNC;
	(* Coordinate System *)
	AxisGroupKin_Inst.In.Target.CoordSys:=KIN_KCS;

	AxisGroupKin_Inst.In.General.Mode := KIN_TARGET_CART;
END_ACTION

ACTION S00_TARGET_CART_P1_action:
AxisGroupKin_Inst.In.Target.Position :=  XYZ_TARG_LIN_CIRC_P1;
END_ACTION

ACTION S10_LIN_XY_P2_entry:
(* Straight line to XYZ_TARG_LIN_CIRC_P2, as soon as XYZ_TARG_LIN_CIRC_P1 has been reached *)

		AxisGroupKin_Inst.In.General.Mode := KIN_LIN_XY;
		AxisGroupKin_Inst.In.Cp.Segment.Position := XYZ_TARG_LIN_CIRC_P2;
(* CP motion parameters *)
		(* settings for whole path / all segments *)
		AxisGroupKin_Inst.In.Cp.Path.VelocityPercentage:=100;
		AxisGroupKin_Inst.In.Cp.Path.FidelityPercentage :=100;
		(* Settings for the segment, which should be added to the queue *)
		AxisGroupKin_Inst.In.Cp.Segment.Translation.Velocity := 1000;
		AxisGroupKin_Inst.In.Cp.Segment.Translation.Acceleration := 100;
		AxisGroupKin_Inst.In.Cp.Segment.Translation.Deceleration := 100;
		AxisGroupKin_Inst.In.Cp.Segment.Translation.Jerk := 100;
		AxisGroupKin_Inst.In.Cp.Segment.Blending.Distance := 50;
		AxisGroupKin_Inst.In.Cp.Segment.Blending.LimitationPercentage := 50;

		AxisGroupKin_Inst.In.Cp.Segment.ID := AxisGroupKin_Inst.In.Cp.Segment.ID + 1;	(* Change the SegmentID to add the segment to the queue *)

		AxisGroupKin_Inst.In.Simu3D.Ctrl.Pen_TCP_WCS := TRUE;
END_ACTION

ACTION S20_CIRC_ZX_Radius_entry:
AxisGroupKin_Inst.In.General.Mode := KIN_CIRC_ZX;
(* Parameters to define the circle *)
AxisGroupKin_Inst.In.Cp.Segment.Circ.Mode := KIN_RADIUS_ANGLE;	(* Define the circle with the radius and angle *)
AxisGroupKin_Inst.In.Cp.Segment.Circ.Direction := KIN_CW;	(* Draw circle ClockWise *)
AxisGroupKin_Inst.In.Cp.Segment.Circ.Radius := XYZ_TARG_LIN_CIRC_R3;
AxisGroupKin_Inst.In.Cp.Segment.Circ.Angle := XYZ_TARG_LIN_CIRC_A3;


AxisGroupKin_Inst.In.Cp.Segment.ID := AxisGroupKin_Inst.In.Cp.Segment.ID + 1;
END_ACTION

ACTION S30_LIN_3D_P4_entry:
AxisGroupKin_Inst.In.General.Mode := KIN_LIN_3D;
AxisGroupKin_Inst.In.Cp.Segment.Position := XYZ_TARG_LIN_CIRC_P4;


AxisGroupKin_Inst.In.Cp.Segment.ID := AxisGroupKin_Inst.In.Cp.Segment.ID + 1;
END_ACTION

ACTION S40_LIN_XY_P1_entry:
AxisGroupKin_Inst.In.General.Mode := KIN_LIN_XY;
AxisGroupKin_Inst.In.Cp.Segment.Position := XYZ_TARG_LIN_CIRC_P1;


AxisGroupKin_Inst.In.Cp.Segment.ID := AxisGroupKin_Inst.In.Cp.Segment.ID + 1;
END_ACTION

ACTION S50_ProgEnd_action:
Done := TRUE;
AxisGroupKin_Inst.In.Simu3D.Ctrl.Pen_TCP_WCS := FALSE;  (* Process Off *)
END_ACTION

TRANSITION Transition:
MC_KinInProximity(Threshold := 0.0,
			Position := AxisGroupKin_Inst.In.Target.Position,
			CoordSys := AxisGroupKin_Inst.In.Target.CoordSys,
			Dimension := 2#0000_0111, ActPos := AxisGroupKin_Inst.Out.General.Position)
AND
AxisGroupKin_Inst.Out.General.Standstill.ActCoordSys
END_TRANSITION

TRANSITION Transition:
(* Wait until the segment was added to the queue; this is not required if FB_KinControl is executed in the same task *)
AxisGroupKin_Inst.Out.Cp.Queue.LastMappedSegID = AxisGroupKin_Inst.In.Cp.Segment.ID
END_TRANSITION

TRANSITION Transition:
(* Wait until the segment was added to the queue; this is not required if FB_KinControl is executed in the same task *)
AxisGroupKin_Inst.Out.Cp.Queue.LastMappedSegID = AxisGroupKin_Inst.In.Cp.Segment.ID
END_TRANSITION

TRANSITION Transition:
(* Wait until the segment was added to the queue; this is not required if FB_KinControl is executed in the same task *)
AxisGroupKin_Inst.Out.Cp.Queue.LastMappedSegID = AxisGroupKin_Inst.In.Cp.Segment.ID
END_TRANSITION

TRANSITION Transition:
(AxisGroupKin_Inst.Out.Cp.Path.EndReached) AND
(AxisGroupKin_Inst.Out.Cp.Queue.LastMappedSegID = AxisGroupKin_Inst.In.Cp.Segment.ID)
END_TRANSITION
END_FUNCTION_BLOCK

(* POU AxisGroupControl_Kinematics/Examples/PRG05_XYZ_FillQueue_LIN3D_with_Array_ST, ST *)
(*##############################################################################################################

	IMPORTANT NOTICE:
 	This example is a special and free service that demonstrates only the basic 
	approach to generating a PLC program as a non-binding sample. 
	SEW is not liable for the contents of the sample program.

	Name:			PRG_XYZ_FillQueue_LIN3D_with_Array_ST
	Job:			Example program			

################################################################################################################*)
FUNCTION_BLOCK PRG05_XYZ_FillQueue_LIN3D_with_Array_ST

VAR_INPUT
	Enable: BOOL;
END_VAR
VAR_OUTPUT
	Active: BOOL;
	Done: BOOL;
END_VAR
VAR
	nState : INT := 0;
	i:INT:=1;
END_VAR
VAR_IN_OUT
	AxisGroupKin_Inst											: ST_AxisGroupKin_Instance;
END_VAR
IF NOT Enable THEN
	Done:=FALSE;
	Active := FALSE;
	i:=1;
	nState:=0;
	RETURN;
END_IF
CASE nState OF
0:	(*Start*)
	IF AxisGroupKin.ConfigDataAvailable THEN
		nState := 5;
	END_IF

5:	(* Initialization and TARGET_CART to last point in queue *)

	(* Initialize kinematics flags*)
	AxisGroupKin_Inst.In.Cp.Settings.PlusTargetCartABC :=FALSE;
	AxisGroupKin_Inst.In.Cp.Settings.UseMasterPosition:=FALSE;

(* CP settings *)
	(* Initialize SegID *)
	AxisGroupKin_Inst.In.Cp.Segment.ID := AxisGroupKin_Inst.Out.Cp.Queue.LastMappedSegID;
	(* Initialize global point array *)
	points[1].x:=10;	points[1].y:=100;	points[1].z:=50;
	points[2].x:=10;	points[2].y:=200;	points[2].z:=100;
	points[3].x:=50;	points[3].y:=300;	points[3].z:=50;
	points[4].x:=100;	points[4].y:=350;	points[4].z:=100;
	points[5].x:=200;	points[5].y:=300;	points[5].z:=50;
	points[6].x:=300;	points[6].y:=200;	points[6].z:=100;
	points[7].x:=300;	points[7].y:=100;	points[7].z:=50;
	points[8].x:=200;	points[8].y:=50;	points[8].z:=100;
	points[9].x:=100;	points[9].y:=10;	points[9].z:=50;
	points[10].x:=50;	points[10].y:=50;	points[10].z:=100;
	(* motion parameters for CP modes *)
	AxisGroupKin_Inst.In.Cp.Segment.Translation.Velocity := 100;
	AxisGroupKin_Inst.In.Cp.Segment.Translation.Acceleration := 100;
	AxisGroupKin_Inst.In.Cp.Segment.Translation.Deceleration := 100;
	AxisGroupKin_Inst.In.Cp.Segment.Translation.Jerk := 100;
	AxisGroupKin_Inst.In.Cp.Segment.Blending.Distance := 30;
	AxisGroupKin_Inst.In.Cp.Segment.Blending.LimitationPercentage := 50;
	AxisGroupKin_Inst.In.Cp.Segment.Mode := KIN_CONTINUOUS_PATH;
	AxisGroupKin_Inst.In.Cp.Path.VelocityPercentage:=100;
	AxisGroupKin_Inst.In.Cp.Path.FidelityPercentage :=100;

(* TARGET_CART settings *)
	(* Set motion parameters for target mode*)
	AxisGroupKin_Inst.In.Target.Cart.Acceleration := CART_ACC50;
	AxisGroupKin_Inst.In.Target.Cart.Deceleration := CART_DEC50;
	AxisGroupKin_Inst.In.Target.Cart.Velocity := CART_VEL50;
	AxisGroupKin_Inst.In.Target.Cart.Jerk:=CART_Jerk100;
	AxisGroupKin_Inst.In.Target.CoordSys := KIN_KCS;
	AxisGroupKin_Inst.In.Target.Synchronization:= KIN_NO_SYNC;
	(* move to last point in array *)
	AxisGroupKin_Inst.In.Target.Position[1] := points[10].x;
	AxisGroupKin_Inst.In.Target.Position[2] := points[10].y;
	AxisGroupKin_Inst.In.Target.Position[3] := points[10].z;

	AxisGroupKin_Inst.In.General.Mode := KIN_TARGET_CART;

	IF (MC_KinInProximity(Threshold := 0.0,
			Position := AxisGroupKin_Inst.In.Target.Position,
			CoordSys := AxisGroupKin_Inst.In.Target.CoordSys,
			Dimension := 2#0000_0111, ActPos := AxisGroupKin_Inst.Out.General.Position)
			AND AxisGroupKin_Inst.Out.General.Standstill.ActCoordSys) THEN
		nState := 10;
	END_IF
10:	(*Fill Queue *)
	IF i <=10 THEN
		AxisGroupKin_Inst.In.Simu3D.Ctrl.Pen_TCP_WCS :=TRUE;
		IF AxisGroupKin_Inst.Out.Cp.Queue.LastMappedSegID = AxisGroupKin_Inst.In.Cp.Segment.ID THEN
			AxisGroupKin_Inst.In.General.Mode := KIN_LIN_3D;
			AxisGroupKin_Inst.In.Cp.Segment.Position[1] := points[i].x;
			AxisGroupKin_Inst.In.Cp.Segment.Position[2] := points[i].y;
			AxisGroupKin_Inst.In.Cp.Segment.Position[3] := points[i].z;
			AxisGroupKin_Inst.In.Cp.Segment.ID := AxisGroupKin_Inst.In.Cp.Segment.ID + 1;
			i:=i+1;
		END_IF
	ELSIF AxisGroupKin_Inst.Out.Cp.Path.EndReached THEN
		Done := TRUE;
		Active := FALSE;
		AxisGroupKin_Inst.In.Simu3D.Ctrl.Pen_TCP_WCS := FALSE;
	END_IF
END_CASE
END_FUNCTION_BLOCK

(* POU AxisGroupControl_Kinematics/Examples/PRG06_XYZ_FillQueue_LIN3D_with_Array_SFC, SFC *)
(*##############################################################################################################

	IMPORTANT NOTICE:
 	This example is a special and free service that demonstrates only the basic 
	approach to generating a PLC program as a non-binding sample. 
	SEW is not liable for the contents of the sample program.

	Name:			PRG_XYZ_FillQueue_LIN3D_with_Array_SFC
	Job:			Example program		

################################################################################################################*)
FUNCTION_BLOCK PRG06_XYZ_FillQueue_LIN3D_with_Array_SFC
VAR_INPUT
	SFCReset:BOOL;
	(*SFCInit:BOOL;*)
	SFCPause:BOOL;

	SFCTipMode:BOOL;
	SFCTip:BOOL;
	SFCEnableLimit:BOOL;
	SFCQuitError:BOOL;

END_VAR
VAR_OUTPUT
	SFCTrans:BOOL;
	SFCError:BOOL;
	SFCErrorStep:STRING;
	SFCErrorPOU:STRING;
	SFCCurrentStep:STRING;
	Done:BOOL;
END_VAR
VAR
	i:INT;
END_VAR
VAR_IN_OUT
	AxisGroupKin_Inst	: ST_AxisGroupKin_Instance;
END_VAR
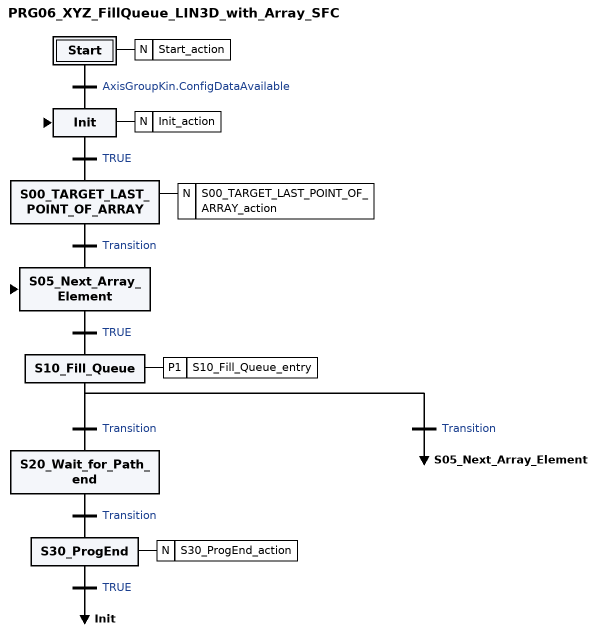
INITIAL_STEP Start:
	Start_action(N);
END_STEP
TRANSITION FROM Start TO Init := AxisGroupKin.ConfigDataAvailable;
END_TRANSITION
STEP Init:
	Init_action(N);
END_STEP
TRANSITION FROM Init TO S00_TARGET_LAST_POINT_OF_ARRAY := TRUE;
END_TRANSITION
STEP S00_TARGET_LAST_POINT_OF_ARRAY:
	S00_TARGET_LAST_POINT_OF_ARRAY_action(N);
END_STEP
TRANSITION FROM S00_TARGET_LAST_POINT_OF_ARRAY TO S05_Next_Array_Element := Transition;
END_TRANSITION
STEP S05_Next_Array_Element:
END_STEP
TRANSITION FROM S05_Next_Array_Element TO S10_Fill_Queue := TRUE;
END_TRANSITION
STEP S10_Fill_Queue:
	S10_Fill_Queue_entry(P1);
END_STEP
TRANSITION FROM S10_Fill_Queue TO S20_Wait_for_Path_end := Transition;
END_TRANSITION
TRANSITION FROM S10_Fill_Queue TO S05_Next_Array_Element := Transition;
END_TRANSITION
STEP S20_Wait_for_Path_end:
END_STEP
TRANSITION FROM S20_Wait_for_Path_end TO S30_ProgEnd := Transition;
END_TRANSITION
STEP S30_ProgEnd:
	S30_ProgEnd_action(N);
END_STEP
TRANSITION FROM S30_ProgEnd TO Init := TRUE;
END_TRANSITION

ACTION Start_action:
Done:=FALSE;
END_ACTION

ACTION Init_action:
(* Initialize kinematics flags*)
	AxisGroupKin_Inst.In.Cp.Settings.PlusTargetCartABC :=FALSE;
	AxisGroupKin_Inst.In.Cp.Settings.UseMasterPosition:=FALSE;

(* CP settings *)
	(* Initialize SegID *)
	AxisGroupKin_Inst.In.Cp.Segment.ID := AxisGroupKin_Inst.Out.Cp.Queue.LastMappedSegID;
	(* Initialize global point array *)
	points[1].x:=10;	points[1].y:=100;	points[1].z:=50;
	points[2].x:=10;	points[2].y:=200;	points[2].z:=100;
	points[3].x:=50;	points[3].y:=300;	points[3].z:=50;
	points[4].x:=100;	points[4].y:=350;	points[4].z:=100;
	points[5].x:=200;	points[5].y:=300;	points[5].z:=50;
	points[6].x:=300;	points[6].y:=200;	points[6].z:=100;
	points[7].x:=300;	points[7].y:=100;	points[7].z:=50;
	points[8].x:=200;	points[8].y:=50;	points[8].z:=100;
	points[9].x:=100;	points[9].y:=10;	points[9].z:=50;
	points[10].x:=50;	points[10].y:=50;	points[10].z:=100;
	(* motion parameters for CP modes *)
	AxisGroupKin_Inst.In.Cp.Segment.Translation.Velocity := 100;
	AxisGroupKin_Inst.In.Cp.Segment.Translation.Acceleration := 100;
	AxisGroupKin_Inst.In.Cp.Segment.Translation.Deceleration := 100;
	AxisGroupKin_Inst.In.Cp.Segment.Translation.Jerk := 100;
	AxisGroupKin_Inst.In.Cp.Segment.Blending.Distance := 30;
	AxisGroupKin_Inst.In.Cp.Segment.Blending.LimitationPercentage := 50;
	AxisGroupKin_Inst.In.Cp.Segment.Mode := KIN_CONTINUOUS_PATH;
	AxisGroupKin_Inst.In.Cp.Path.VelocityPercentage:=100;
	AxisGroupKin_Inst.In.Cp.Path.FidelityPercentage :=100;

(* TARGET_CART settings *)
	(* Set motion parameters for target mode*)
	AxisGroupKin_Inst.In.Target.Cart.Acceleration := CART_ACC50;
	AxisGroupKin_Inst.In.Target.Cart.Deceleration := CART_DEC50;
	AxisGroupKin_Inst.In.Target.Cart.Velocity := CART_VEL50;
	AxisGroupKin_Inst.In.Target.Cart.Jerk:=CART_Jerk100;
	AxisGroupKin_Inst.In.Target.CoordSys := KIN_KCS;
	AxisGroupKin_Inst.In.Target.Synchronization:= KIN_NO_SYNC;

	AxisGroupKin_Inst.In.General.Mode := KIN_TARGET_CART;

	i:=1;
END_ACTION

ACTION S00_TARGET_LAST_POINT_OF_ARRAY_action:
(* move to last point in array *)
AxisGroupKin_Inst.In.Target.Position[1] := points[10].x;
AxisGroupKin_Inst.In.Target.Position[2] := points[10].y;
AxisGroupKin_Inst.In.Target.Position[3] := points[10].z;
END_ACTION

ACTION S10_Fill_Queue_entry:
AxisGroupKin_Inst.In.General.Mode			:= KIN_LIN_3D;
AxisGroupKin_Inst.In.Cp.Segment.Position[1]	:= points[i].x;
AxisGroupKin_Inst.In.Cp.Segment.Position[2] 	:= points[i].y;
AxisGroupKin_Inst.In.Cp.Segment.Position[3] 	:= points[i].z;
AxisGroupKin_Inst.In.Cp.Segment.ID 		:= AxisGroupKin_Inst.In.Cp.Segment.ID + 1;

i:=i+1;
END_ACTION

ACTION S30_ProgEnd_action:
Done:=TRUE;
END_ACTION

TRANSITION Transition:
MC_KinInProximity(Threshold := 0.0,
			Position := AxisGroupKin_Inst.In.Target.Position,
			CoordSys := AxisGroupKin_Inst.In.Target.CoordSys,
			Dimension := 2#0000_0111, ActPos := AxisGroupKin_Inst.Out.General.Position)

AND
AxisGroupKin_Inst.Out.General.Standstill.ActCoordSys
END_TRANSITION

TRANSITION Transition:
(AxisGroupKin_Inst.Out.Cp.Queue.LastMappedSegID= AxisGroupKin_Inst.In.Cp.Segment.ID) AND (i >10)
END_TRANSITION

TRANSITION Transition:
AxisGroupKin_Inst.Out.Cp.Queue.LastMappedSegID = AxisGroupKin_Inst.In.Cp.Segment.ID
END_TRANSITION

TRANSITION Transition:
AxisGroupKin_Inst.Out.Cp.Path.EndReached
END_TRANSITION
END_FUNCTION_BLOCK

(* POU AxisGroupControl_Kinematics/Examples/PRG07_XYZ_USER_ST, ST *)
(*##############################################################################################################

	IMPORTANT NOTICE:
 	This example is a special and free service that demonstrates only the basic 
	approach to generating a PLC program as a non-binding sample. 
	SEW is not liable for the contents of the sample program.

	Name:			PRG_XYZ_USER_ST
	Job:			Example program
					Simple program, in which you can implement your own sample sequence.			

################################################################################################################*)
FUNCTION_BLOCK PRG07_XYZ_USER_ST
VAR_INPUT
	Enable : BOOL;
END_VAR
VAR_OUTPUT
	Active : BOOL;
	Done : BOOL;
END_VAR
VAR
	nState : INT;
	fbRtrig : R_TRIG;
END_VAR
VAR_IN_OUT
	AxisGroupKin_Inst											: ST_AxisGroupKin_Instance;
END_VAR
(* Initialisation at rising edge of VAR_INPUT Enable *)
fbRtrig(CLK:=Enable);
IF fbRtrig.Q THEN
	nState	:= 0;
	Active := TRUE;
END_IF

(* No execution, if Enable = False *)
IF NOT Enable THEN
	Done := FALSE;
	RETURN;
END_IF

CASE nState OF
0:	(*Start*)
	IF AxisGroupKin.ConfigDataAvailable THEN
		nState := 5;
	END_IF
5:	(* TARGET_CART to XYZ_USER_P1 *)
	(* Initialize Kinematic Flags*)
	AxisGroupKin_Inst.In.Cp.Settings.PlusTargetCartABC:=FALSE;
	AxisGroupKin_Inst.In.Cp.Settings.UseMasterPosition:=FALSE;

(* TARGET_CART settings *)
	(* Motion Parameters *)
	AxisGroupKin_Inst.In.Target.Cart.Velocity := CART_VEL50;
	AxisGroupKin_Inst.In.Target.Cart.Acceleration := CART_ACC50;
	AxisGroupKin_Inst.In.Target.Cart.Deceleration := CART_DEC50;
	AxisGroupKin_Inst.In.Target.Cart.Jerk:=CART_Jerk100;
	AxisGroupKin_Inst.In.Target.Synchronization:= KIN_NO_SYNC;
	(* Coordinate System *)
	AxisGroupKin_Inst.In.Target.CoordSys:=KIN_KCS;

	AxisGroupKin_Inst.In.General.Mode := KIN_TARGET_CART;

	AxisGroupKin_Inst.In.Simu3D.Ctrl.Pen_TCP_WCS := TRUE;  (* Process On *)

	AxisGroupKin_Inst.In.Target.Position := XYZ_USER_P1;
	IF (MC_KinInProximity(Threshold := 0.0,
			Position := AxisGroupKin_Inst.In.Target.Position,
			CoordSys := AxisGroupKin_Inst.In.Target.CoordSys,
			Dimension := 2#0000_0111, ActPos := AxisGroupKin_Inst.Out.General.Position)
			AND AxisGroupKin_Inst.Out.General.Standstill.ActCoordSys) THEN
		nState := 10;
	END_IF

10:	(* TARGET_CART to XYZ_USER_P2 *)
	AxisGroupKin_Inst.In.Target.Position := XYZ_USER_P2;
	IF (MC_KinInProximity(Threshold := 0.0,
			Position := AxisGroupKin_Inst.In.Target.Position,
			CoordSys := AxisGroupKin_Inst.In.Target.CoordSys,
			Dimension := 2#0000_0111, ActPos := AxisGroupKin_Inst.Out.General.Position)
			AND AxisGroupKin_Inst.Out.General.Standstill.ActCoordSys) THEN
		Done := TRUE;
		Active := FALSE;
		AxisGroupKin_Inst.In.Simu3D.Ctrl.Pen_TCP_WCS := FALSE;  (* Process Off *)
	END_IF

ELSE
;

END_CASE
END_FUNCTION_BLOCK

(* POU AxisGroupControl_Kinematics/Examples/PRG08_XYZ_USER_SFC, SFC *)
(*##############################################################################################################

	IMPORTANT NOTICE:
 	This example is a special and free service that demonstrates only the basic 
	approach to generating a PLC program as a non-binding sample. 
	SEW is not liable for the contents of the sample program.

	Name:			PRG_XYZ_USER_SFC
	Job:			Example program
					Simple program, in which you can implement your own sample sequence.				

################################################################################################################*)
FUNCTION_BLOCK PRG08_XYZ_USER_SFC
VAR_INPUT
	SFCReset:BOOL;
	(*SFCInit:BOOL;*)
	SFCPause:BOOL;

	SFCTipMode:BOOL;
	SFCTip:BOOL;
	SFCEnableLimit:BOOL;
	SFCQuitError:BOOL;

END_VAR
VAR_OUTPUT
	SFCTrans:BOOL;
	SFCError:BOOL;
	SFCErrorStep:STRING;
	SFCErrorPOU:STRING;
(*	SFCErrorAnalyzation:STRING;*)
	SFCCurrentStep:STRING;
	Done:BOOL;
END_VAR
VAR

END_VAR
VAR_IN_OUT
	AxisGroupKin_Inst											: ST_AxisGroupKin_Instance;
END_VAR
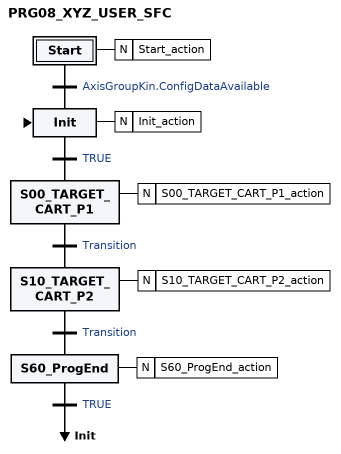
INITIAL_STEP Start:
	Start_action(N);
END_STEP
TRANSITION FROM Start TO Init := AxisGroupKin.ConfigDataAvailable;
END_TRANSITION
STEP Init:
	Init_action(N);
END_STEP
TRANSITION FROM Init TO S00_TARGET_CART_P1 := TRUE;
END_TRANSITION
STEP S00_TARGET_CART_P1:
	S00_TARGET_CART_P1_action(N);
END_STEP
TRANSITION FROM S00_TARGET_CART_P1 TO S10_TARGET_CART_P2 := Transition;
END_TRANSITION
STEP S10_TARGET_CART_P2:
	S10_TARGET_CART_P2_action(N);
END_STEP
TRANSITION FROM S10_TARGET_CART_P2 TO S60_ProgEnd := Transition;
END_TRANSITION
STEP S60_ProgEnd:
	S60_ProgEnd_action(N);
END_STEP
TRANSITION FROM S60_ProgEnd TO Init := TRUE;
END_TRANSITION

ACTION Start_action:
Done:=FALSE;
END_ACTION

ACTION Init_action:
(* Initialize Kinematic Flags*)
AxisGroupKin_Inst.In.Cp.Settings.PlusTargetCartABC:=FALSE;
AxisGroupKin_Inst.In.Cp.Settings.UseMasterPosition:=FALSE;

(* TARGET_CART settings *)
	(* Motion Parameters *)
	AxisGroupKin_Inst.In.Target.Cart.Velocity := CART_VEL50;
	AxisGroupKin_Inst.In.Target.Cart.Acceleration := CART_ACC50;
	AxisGroupKin_Inst.In.Target.Cart.Deceleration := CART_DEC50;
	AxisGroupKin_Inst.In.Target.Cart.Jerk:=CART_Jerk100;
	AxisGroupKin_Inst.In.Target.Synchronization:= KIN_NO_SYNC;
	(* Coordinate System *)
	AxisGroupKin_Inst.In.Target.CoordSys:=KIN_KCS;

AxisGroupKin_Inst.In.General.Mode := KIN_TARGET_CART;

AxisGroupKin_Inst.In.Simu3D.Ctrl.Pen_TCP_WCS := TRUE;  (* Process On *)
END_ACTION

ACTION S00_TARGET_CART_P1_action:
AxisGroupKin_Inst.In.Target.Position := XYZ_USER_P1;
END_ACTION

ACTION S10_TARGET_CART_P2_action:
AxisGroupKin_Inst.In.Target.Position := XYZ_USER_P2;
END_ACTION

ACTION S60_ProgEnd_action:
Done := TRUE;
AxisGroupKin_Inst.In.Simu3D.Ctrl.Pen_TCP_WCS := FALSE;  (* Process Off *)
END_ACTION

TRANSITION Transition:
MC_KinInProximity(Threshold := 0.0,
			Position := AxisGroupKin_Inst.In.Target.Position,
			CoordSys := AxisGroupKin_Inst.In.Target.CoordSys,
			Dimension := 2#0000_0111, ActPos := AxisGroupKin_Inst.Out.General.Position)
AND
AxisGroupKin_Inst.Out.General.Standstill.ActCoordSys
END_TRANSITION

TRANSITION Transition:
MC_KinInProximity(Threshold := 0.0,
			Position := AxisGroupKin_Inst.In.Target.Position,
			CoordSys := AxisGroupKin_Inst.In.Target.CoordSys,
			Dimension := 2#0000_0111, ActPos := AxisGroupKin_Inst.Out.General.Position)
AND
AxisGroupKin_Inst.Out.General.Standstill.ActCoordSys
END_TRANSITION
END_FUNCTION_BLOCK

(* POU PRG_Kinematics/PRG_TaskPriority_Kinematics, ST *)
PROGRAM PRG_TaskPriority_Kinematics
VAR
END_VAR
(*#######################################################################################

	PRG_TaskPriority_Kinematics

	ToDo: Call this program in the task configuration after PRG_TaskPriority();

########################################################################################*)

(* Do not remove! *)
AxisGroupControl_Priority_Kinematics();
END_PROGRAM

(* POU SewRobotLanguage/FB_SewRobotLanguage_User_Function, ST *)
(*##############################################################################################################

	IMPORTANT NOTICE:
 	This example is a special and free service that demonstrates only the basic 
	approach to generating a PLC program as a non-binding sample. 
	SEW is not liable for the contents of the sample program.

	Name:			FB_SewRobotLanguage_User_Function
	Job:			Contains User Functions that can be called in SRL Program

################################################################################################################*)
FUNCTION_BLOCK FB_SewRobotLanguage_User_Function
VAR_INPUT
	Enable								: BOOL;				(* Enable of Function*)
	NumberOfFunction				: INT;					(* Number of the Fuction what will be executed*)
	bParaValue						: BOOL;				(* Boolean	Value *)
	rParaValue						: LREAL;				(* Real 	Value *)
	posParaValue						: ST_SRL_DimPos; 	(* Position Vektor *)
	Instance							: UINT;
END_VAR
VAR_OUTPUT
	Done								: BOOL;				(* true if function is executed correctly*)
	Error								: BOOL;				(* Error Flag*)
	ErrorID								: DWORD;				(* Error ID*)
END_VAR
VAR_IN_OUT
	SRL_Dat_Var						: ST_SRL_Variables;
	AxisGroupKin_Inst				: ST_AxisGroupKin_Instance;	(*AxisGroupControl Kinematics Variable*)
END_VAR
VAR
	(*Handling Kin: Zuweisung Dynamikwerte anhand der SegParRecords*)
	nIndex 								: UINT;


	SegParaRecCart_Act				: UINT;
	SegParaRecAxis_Act				: UINT;
	SegParaRecCp_Act				: UINT;
	SegParaRecRot_Act				: UINT;
	SegParaRecTp_Act				: UINT;

	nSynchronization					: WORD;

	fbTON					: TON;
	tTime					: TIME;

	ModuleName 			: STRING(50)		:='SRL_User_Function';
	Message				: STRING(128)	:='SRL_User_Function';
	nTaskID				: WORD;
	nTaskPriority			: DINT;
END_VAR
IF ((Instance < 1) OR (Instance > KIN_AXISGROUPKIN_MAX_NUMBER_OF_KINEMATICS_INSTANCES)) THEN
	MC_MsgHandler_Enter(
		Class 		:= MSGHANDLER_CLASS_ERROR,
		Source 	:= MSGHANDLER_SOURCE_TECHNOLOGYMODULE,
		Module 	:= 'SewRobotLanguage',
		Instance 	:= Instance,
		ID 			:= E_KIN_SRL_INSTANCENUMBER_NOT_VALID,
		Text 		:= 'MC_Enter_Message_Buffer_SRL: InstanceNumber Not Valid',
		Value_n1 	:= 0 ,
		Value_n2 	:= 0,
		Value_f1 	:= 0,
		Value_f2 	:= 0,
		ErrorArchivingOnlyAfterReset := FALSE,
		ForceEntryInNewElement := FALSE);
		(*weil kein gültige Instanznummer da, hier die 1 auf Fehler setzen*)
		SRL.Inst[1].Interface.Out.FBError	:= TRUE;
		SRL.Inst[1].Interface.Out.FBErrorID	:= E_KIN_SRL_INSTANCENUMBER_NOT_VALID;

	RETURN;
END_IF

tTime:=REAL_TO_TIME(rParaValue);

fbTON(IN:=Enable , PT:=tTime );

IF Enable THEN
	CASE NumberOfFunction OF
		11:(* SegParRecAxis *)

			SegParaRecAxis_Act := LREAL_TO_UINT(rParaValue);
			IF (SegParaRecAxis_Act > 8) OR (SegParaRecAxis_Act < 1) THEN(*tbd ID festlegen*)
				Message:= ' SegParRecord Number §n1§ not valid => Init Program and Reset Error';
				MC_Enter_Message_Buffer_HandlingKin(
					E_HANDLINGKIN_SEG_PAR_RECORD_NUMBER_NOT_VALID,Message,0,0,0,0,TRUE,Instance,Error,ErrorID);
				RETURN;
			END_IF
			FOR nIndex := 1 TO 8 DO
				(*Es wird nur noch die Geschwindigkeit vom Override Percentage beeinflußt *)

				SRL_Dat_Var.PositionData.Value[SRL_SYS_IN_AXIS_VEL].Dim[nIndex]:=AxisGroupHandlingKin.Inst[Instance].Config.SegmentParameterRecord[SegParaRecAxis_Act].AxisVel[nIndex];
				SRL_Dat_Var.PositionData.Value[SRL_SYS_IN_AXIS_ACC].Dim[nIndex]:=AxisGroupHandlingKin.Inst[Instance].Config.SegmentParameterRecord[SegParaRecAxis_Act].AxisAcc[nIndex]		(** TargetVelocityPercentagefaktor*TargetVelocityPercentagefaktor*);
				SRL_Dat_Var.PositionData.Value[SRL_SYS_IN_AXIS_DEC].Dim[nIndex]:=AxisGroupHandlingKin.Inst[Instance].Config.SegmentParameterRecord[SegParaRecAxis_Act].AxisDec[nIndex]		(** TargetVelocityPercentagefaktor*TargetVelocityPercentagefaktor*);
				IF AxisGroupKin_Inst.Config.General.RealJerk_InsteadOfJerkTime THEN
					SRL_Dat_Var.PositionData.Value[SRL_SYS_IN_AXIS_JERK].Dim[nIndex]:=AxisGroupHandlingKin.Inst[Instance].Config.SegmentParameterRecord[SegParaRecAxis_Act].AxisJerk[nIndex](** TargetVelocityPercentagefaktor*TargetVelocityPercentagefaktor*TargetVelocityPercentagefaktor*);
				ELSE
					SRL_Dat_Var.PositionData.Value[SRL_SYS_IN_AXIS_JERK].Dim[nIndex]:=AxisGroupHandlingKin.Inst[Instance].Config.SegmentParameterRecord[SegParaRecAxis_Act].AxisJerk[nIndex] (*/ TargetVelocityPercentagefaktor*)	;
				END_IF
			END_FOR
			nSynchronization:=0;
			nSynchronization.1:= AxisGroupHandlingKin.Inst[Instance].Config.SegmentParameterRecord[SegParaRecAxis_Act].AxisSynchronization[1];
			nSynchronization.2:= AxisGroupHandlingKin.Inst[Instance].Config.SegmentParameterRecord[SegParaRecAxis_Act].AxisSynchronization[2];
			nSynchronization.3:= AxisGroupHandlingKin.Inst[Instance].Config.SegmentParameterRecord[SegParaRecAxis_Act].AxisSynchronization[3];
			nSynchronization.4:= AxisGroupHandlingKin.Inst[Instance].Config.SegmentParameterRecord[SegParaRecAxis_Act].AxisSynchronization[4];
			nSynchronization.5:= AxisGroupHandlingKin.Inst[Instance].Config.SegmentParameterRecord[SegParaRecAxis_Act].AxisSynchronization[5];
			nSynchronization.6:= AxisGroupHandlingKin.Inst[Instance].Config.SegmentParameterRecord[SegParaRecAxis_Act].AxisSynchronization[6];
			nSynchronization.7:= AxisGroupHandlingKin.Inst[Instance].Config.SegmentParameterRecord[SegParaRecAxis_Act].AxisSynchronization[7];
			nSynchronization.8:= AxisGroupHandlingKin.Inst[Instance].Config.SegmentParameterRecord[SegParaRecAxis_Act].AxisSynchronization[8];
			SRL_Dat_Var.RealData.Value[SRL_SYS_IN_TARGET_AXIS_SYNC]:=WORD_TO_LREAL(nSynchronization);
			Done:=TRUE;

		12:(* SegParRecCart	*)

			SegParaRecCart_Act:=LREAL_TO_UINT(rParaValue);
			IF (SegParaRecCart_Act > 8) OR (SegParaRecCart_Act < 1) THEN(*tbd ID festlegen*)
				Message:= ' SegParRecord Number §n1§ not valid => Init Program and Reset Error';
				MC_Enter_Message_Buffer_HandlingKin(
					E_HANDLINGKIN_SEG_PAR_RECORD_NUMBER_NOT_VALID,Message,0,0,0,0,TRUE,Instance,Error,ErrorID);
				RETURN;
			END_IF
			FOR nIndex := 1 TO 6 DO
				SRL_Dat_Var.PositionData.Value[SRL_SYS_IN_CART_VEL].Dim[nIndex]:=AxisGroupHandlingKin.Inst[Instance].Config.SegmentParameterRecord[SegParaRecCart_Act].CartVel[nIndex]	;
				SRL_Dat_Var.PositionData.Value[SRL_SYS_IN_CART_ACC].Dim[nIndex]:=AxisGroupHandlingKin.Inst[Instance].Config.SegmentParameterRecord[SegParaRecCart_Act].CartAcc[nIndex]	(** TargetVelocityPercentagefaktor*TargetVelocityPercentagefaktor*);
				SRL_Dat_Var.PositionData.Value[SRL_SYS_IN_CART_DEC].Dim[nIndex]:=AxisGroupHandlingKin.Inst[Instance].Config.SegmentParameterRecord[SegParaRecCart_Act].CartDec[nIndex]	(** TargetVelocityPercentagefaktor*TargetVelocityPercentagefaktor*);
				IF AxisGroupKin_Inst.Config.General.RealJerk_InsteadOfJerkTime THEN
					SRL_Dat_Var.PositionData.Value[SRL_SYS_IN_CART_JERK].Dim[nIndex]:=AxisGroupHandlingKin.Inst[Instance].Config.SegmentParameterRecord[SegParaRecCart_Act].CartJerk[nIndex](* / (TargetVelocityPercentagefaktor * TargetVelocityPercentagefaktor *TargetVelocityPercentagefaktor )*);
				ELSE
					SRL_Dat_Var.PositionData.Value[SRL_SYS_IN_CART_JERK].Dim[nIndex]:=AxisGroupHandlingKin.Inst[Instance].Config.SegmentParameterRecord[SegParaRecCart_Act].CartJerk[nIndex] (* / (TargetVelocityPercentagefaktor )*);
				END_IF
			END_FOR

			(* Werte für Achse7 und Achse 8 auch in Callf12 übernehmen, damit die Zusatzachsen in Programm Nr.4 auch korrekt verfahren werden können.  *)
			FOR nIndex := 7 TO 8 DO
				SRL_Dat_Var.PositionData.Value[SRL_SYS_IN_AXIS_VEL].Dim[nIndex]:=AxisGroupHandlingKin.Inst[Instance].Config.SegmentParameterRecord[SegParaRecCart_Act].AxisVel[nIndex];
				SRL_Dat_Var.PositionData.Value[SRL_SYS_IN_AXIS_ACC].Dim[nIndex]:=AxisGroupHandlingKin.Inst[Instance].Config.SegmentParameterRecord[SegParaRecCart_Act].AxisAcc[nIndex]	;
				SRL_Dat_Var.PositionData.Value[SRL_SYS_IN_AXIS_DEC].Dim[nIndex]:=AxisGroupHandlingKin.Inst[Instance].Config.SegmentParameterRecord[SegParaRecCart_Act].AxisDec[nIndex];
				IF AxisGroupKin_Inst.Config.General.RealJerk_InsteadOfJerkTime THEN
					SRL_Dat_Var.PositionData.Value[SRL_SYS_IN_AXIS_JERK].Dim[nIndex]:=AxisGroupHandlingKin.Inst[Instance].Config.SegmentParameterRecord[SegParaRecCart_Act].AxisJerk[nIndex];
				ELSE
					SRL_Dat_Var.PositionData.Value[SRL_SYS_IN_AXIS_JERK].Dim[nIndex]:=AxisGroupHandlingKin.Inst[Instance].Config.SegmentParameterRecord[SegParaRecCart_Act].AxisJerk[nIndex];
				END_IF
			END_FOR

			(*Die Synchronisation liegt Bitweise vor. Allerdings ist im SegParRecord eine Sync für:
				- die Achsweise Interpolation vorgesehen und
				- für die Cartesische Interpolation vorgesehen.
			In der Kin Schnittstelle gibt es aber nur einen Wert für die Synchronisation, der für Target Axes und Target Cart gilt.
			Deshalb wird Abhängigkeit vom Kin-Mode die Synchronisation kopiert*)

			nSynchronization:=0;
			nSynchronization.1:= AxisGroupHandlingKin.Inst[Instance].Config.SegmentParameterRecord[SegParaRecCart_Act].CartSynchronization[1];
			nSynchronization.2:= AxisGroupHandlingKin.Inst[Instance].Config.SegmentParameterRecord[SegParaRecCart_Act].CartSynchronization[2];
			nSynchronization.3:= AxisGroupHandlingKin.Inst[Instance].Config.SegmentParameterRecord[SegParaRecCart_Act].CartSynchronization[3];
			nSynchronization.4:= AxisGroupHandlingKin.Inst[Instance].Config.SegmentParameterRecord[SegParaRecCart_Act].CartSynchronization[4];
			nSynchronization.5:= AxisGroupHandlingKin.Inst[Instance].Config.SegmentParameterRecord[SegParaRecCart_Act].CartSynchronization[5];
			nSynchronization.6:= AxisGroupHandlingKin.Inst[Instance].Config.SegmentParameterRecord[SegParaRecCart_Act].CartSynchronization[6];
			SRL_Dat_Var.RealData.Value[SRL_SYS_IN_TARGET_CART_SYNC]:=WORD_TO_LREAL(nSynchronization);
			Done:=TRUE;

		13:(* SegParRecCp	*)

			SegParaRecCp_Act:=LREAL_TO_UINT(rParaValue);
			IF (SegParaRecCp_Act > 8) OR (SegParaRecCp_Act < 1) THEN
				Message:= ' SegParRecord Number §n1§ not valid => Init Program and Reset Error';
				MC_Enter_Message_Buffer_HandlingKin(
					E_HANDLINGKIN_SEG_PAR_RECORD_NUMBER_NOT_VALID,Message,0,0,0,0,TRUE,Instance,Error,ErrorID);
				RETURN;
			END_IF
			SRL_Dat_Var.RealData.Value[SRL_SYS_IN_CP_VEL]		:=AxisGroupHandlingKin.Inst[Instance].Config.SegmentParameterRecord[SegParaRecCp_Act].TransVel;
			SRL_Dat_Var.RealData.Value[SRL_SYS_IN_CP_ACC]		:=AxisGroupHandlingKin.Inst[Instance].Config.SegmentParameterRecord[SegParaRecCp_Act].TransAcc;
			SRL_Dat_Var.RealData.Value[SRL_SYS_IN_CP_DEC]		:=AxisGroupHandlingKin.Inst[Instance].Config.SegmentParameterRecord[SegParaRecCp_Act].TransDec;
			SRL_Dat_Var.RealData.Value[SRL_SYS_IN_CP_JERK]		:=AxisGroupHandlingKin.Inst[Instance].Config.SegmentParameterRecord[SegParaRecCp_Act].TransJerk;

			SRL_Dat_Var.RealData.Value[SRL_SYS_IN_CP_BLENDING_LIMITATION_PERC]	:=AxisGroupHandlingKin.Inst[Instance].Config.SegmentParameterRecord[SegParaRecCp_Act].BlendingLimitationPercentage;
			SRL_Dat_Var.RealData.Value[SRL_SYS_IN_CP_BLENDING_VEL_PERC]			:=AxisGroupHandlingKin.Inst[Instance].Config.SegmentParameterRecord[SegParaRecCp_Act].BlendingVelocityPercentage;
			SRL_Dat_Var.RealData.Value[SRL_SYS_IN_CP_BLENDING_VEL_PROFILE]		:=AxisGroupHandlingKin.Inst[Instance].Config.SegmentParameterRecord[SegParaRecCp_Act].BlendingVelocityProfile;
			Done:=TRUE;

		14:(*SegParRecRot	*)

			SegParaRecRot_Act:=LREAL_TO_UINT(rParaValue);
			(*Die SRL_SYS_IN_ROT_BLENDING_DISTANCE  für die Orientierung wird aus dem angewählten SegParaRecRot_Act  entnommen
				=> damit kann im Programm über die HandlingKinSysVar SegParRec_Rot der SegParRec ausgewählt werden aus dem die RotBlendingDist 
					entnommen werden soll*)
			IF (SegParaRecRot_Act > 8) OR (SegParaRecRot_Act < 1) THEN(*tbd ID festlegen*)
				Message:= ' SegParRecord Number §n1§ not valid => Init Program and Reset Error';
				MC_Enter_Message_Buffer_HandlingKin(
					E_HANDLINGKIN_SEG_PAR_RECORD_NUMBER_NOT_VALID,Message,0,0,0,0,TRUE,Instance,Error,ErrorID);
				RETURN;
			END_IF
			SRL_Dat_Var.RealData.Value[SRL_SYS_IN_ROT_BLENDING_DISTANCE] := AxisGroupHandlingKin.Inst[Instance].Config.SegmentParameterRecord[SegParaRecRot_Act].RotBlendingDistance;
			Done:=TRUE;

		15:(*SegParRec_Tp	*)

			SegParaRecTp_Act:=LREAL_TO_UINT(rParaValue);
			(*Die SRL_SYS_IN_TP_REMAINING_DISTANCE  für den Restweg wird aus dem angewählten  SegParaRecRot_Act  entnommen
				zusätzlich wird mit dem RemainingDistancePercentage/100 multipliziert
				=> damit kann im Programm über die HandlingKinSysVar SegParRec_Tp der SegParRec ausgewählt werden aus dem die SRL_SYS_IN_TP_REMAINING_DISTANCE 
					entnommen werden soll*)
			IF (SegParaRecTp_Act > 8) OR (SegParaRecTp_Act < 1) THEN(*tbd ID festlegen*)
				Message:= ' SegParRecord Number §n1§ not valid => Init Program and Reset Error';
				MC_Enter_Message_Buffer_HandlingKin(
					E_HANDLINGKIN_SEG_PAR_RECORD_NUMBER_NOT_VALID,Message,0,0,0,0,TRUE,Instance,Error,ErrorID);
				RETURN;
			END_IF
			SRL_Dat_Var.RealData.Value[SRL_SYS_IN_TP_REMAINING_DISTANCE] := (AxisGroupHandlingKin.Inst[Instance].Config.SegmentParameterRecord[SegParaRecTp_Act].RemainingDistance
																										 * (AxisGroupHandlingKinProfile.Inst[Instance].Standard.In.PrgControlAdditional.RemainingDistancePercentage/100.0));
			(*Die Dynamikwerte werden aus dem gleichen SegParRecord entnommen wie die distance*)
			FOR nIndex := 1 TO 6 DO
				SRL_Dat_Var.PositionData.Value[SRL_SYS_IN_CART_TP_VEL].Dim[nIndex]:=AxisGroupHandlingKin.Inst[Instance].Config.SegmentParameterRecord[SegParaRecTp_Act].CartVel[nIndex];
				SRL_Dat_Var.PositionData.Value[SRL_SYS_IN_CART_TP_ACC].Dim[nIndex]:=AxisGroupHandlingKin.Inst[Instance].Config.SegmentParameterRecord[SegParaRecTp_Act].CartAcc[nIndex]	(** TargetVelocityPercentagefaktor*TargetVelocityPercentagefaktor*);
				SRL_Dat_Var.PositionData.Value[SRL_SYS_IN_CART_TP_DEC].Dim[nIndex]:=AxisGroupHandlingKin.Inst[Instance].Config.SegmentParameterRecord[SegParaRecTp_Act].CartDec[nIndex]	(** TargetVelocityPercentagefaktor*TargetVelocityPercentagefaktor*);
				IF AxisGroupKin_Inst.Config.General.RealJerk_InsteadOfJerkTime THEN
					SRL_Dat_Var.PositionData.Value[SRL_SYS_IN_CART_TP_JERK].Dim[nIndex]:=AxisGroupHandlingKin.Inst[Instance].Config.SegmentParameterRecord[SegParaRecTp_Act].CartJerk[nIndex](* / (TargetVelocityPercentagefaktor * TargetVelocityPercentagefaktor *TargetVelocityPercentagefaktor )*);
				ELSE
					SRL_Dat_Var.PositionData.Value[SRL_SYS_IN_CART_TP_JERK].Dim[nIndex]:=AxisGroupHandlingKin.Inst[Instance].Config.SegmentParameterRecord[SegParaRecTp_Act].CartJerk[nIndex] (* / (TargetVelocityPercentagefaktor )*);
				END_IF
			END_FOR
			Done:=TRUE;

		1:
				Done:=fbTON.Q;
		2:
				Done:=TRUE;
		3:
				Done:=TRUE;
		4:
				Done:=TRUE;
		5:
				Done:=TRUE;
		6:
				Done:=TRUE;
		7:
				Done:=TRUE;
		8:
				Done:=TRUE;
		9:
				Done:=TRUE;
		10:
				Done:=TRUE;


	ELSE
		(* -------------Error--------------------*)
		Message:=CONCAT('Function Number : ',INT_TO_STRING(NumberOfFunction) );
		Message:=CONCAT(Message,' is not valid');
		MC_Enter_Message_Buffer_SRL(E_KIN_SRL_FUNCTION_NUMBER_NOT_VALID,  Message, 0, 0, 0, 0,TRUE, Instance, Error, ErrorID);
	END_CASE
ELSE
	Done	:=FALSE;
END_IF
END_FUNCTION_BLOCK
